C05384=1030.378,261.013,-119.631,170.542,45.453,158.713
C05385=1030.370,260.765,-119.601,170.539,45.453,158.712
C05386=1030.364,260.517,-119.572,170.535,45.454,158.712
C05387=1030.357,260.269,-119.542,170.532,45.455,158.712
C05388=1030.351,260.021,-119.513,170.528,45.456,158.712
C05389=1030.344,259.773,-119.483,170.525,45.457,158.712
C05390=1030.337,259.524,-119.453,170.521,45.457,158.711
C05391=1030.330,259.277,-119.424,170.518,45.458,158.711
C05392=1030.323,259.028,-119.395,170.513,45.459,158.711
C05393=1030.316,258.780,-119.366,170.510,45.460,158.711
C05394=1030.309,258.531,-119.336,170.506,45.461,158.711
C05395=1030.303,258.283,-119.307,170.503,45.461,158.710
C05396=1030.295,258.035,-119.277,170.499,45.462,158.710
C05397=1030.289,257.787,-119.248,170.496,45.463,158.710
C05398=1030.282,257.538,-119.219,170.492,45.464,158.710
C05399=1030.275,257.291,-119.189,170.489,45.465,158.710
C05400=1030.269,257.042,-119.159,170.485,45.466,158.709
C05401=1030.262,256.794,-119.130,170.482,45.466,158.709
C05402=1030.255,256.547,-119.101,170.478,45.467,158.709
C05403=1030.248,256.298,-119.072,170.475,45.468,158.709
C05404=1030.242,256.050,-119.043,170.471,45.469,158.709
C05405=1030.235,255.802,-119.013,170.468,45.470,158.709
C05406=1030.229,255.553,-118.984,170.465,45.470,158.708
C05407=1030.221,255.305,-118.955,170.461,45.471,158.708
C05408=1030.215,255.057,-118.926,170.458,45.472,158.708
C05409=1030.208,254.809,-118.896,170.454,45.473,158.708
C05410=1030.201,254.560,-118.867,170.451,45.474,158.708
C05411=1030.195,254.312,-118.838,170.447,45.475,158.708
C05412=1030.187,254.064,-118.809,170.444,45.476,158.707
C05413=1030.181,253.816,-118.780,170.440,45.477,158.707
C05414=1030.175,253.568,-118.750,170.437,45.478,158.707
C05415=1030.168,253.319,-118.721,170.434,45.478,158.707
C05416=1030.162,253.071,-118.691,170.430,45.479,158.707
C05417=1030.155,252.823,-118.663,170.427,45.480,158.706
C05418=1030.148,252.575,-118.634,170.423,45.481,158.706
C05419=1030.141,252.326,-118.605,170.420,45.482,158.706
C05420=1030.135,252.078,-118.576,170.417,45.483,158.706
C05421=1030.128,251.830,-118.545,170.413,45.484,158.706
C05422=1030.121,251.582,-118.517,170.410,45.484,158.706
C05423=1030.115,251.334,-118.488,170.406,45.485,158.705
C05424=1030.108,251.085,-118.459,170.403,45.486,158.705
C05425=1030.102,250.837,-118.429,170.400,45.487,158.705
C05426=1030.095,250.589,-118.400,170.396,45.488,158.705
C05427=1030.088,250.341,-118.372,170.393,45.489,158.705
C05428=1030.082,250.092,-118.343,170.389,45.490,158.705
C05429=1030.075,249.844,-118.314,170.386,45.491,158.704
C05430=1030.069,249.596,-118.284,170.383,45.491,158.704
C05431=1030.059,249.229,-118.242,170.378,45.493,158.704
C05432=1030.049,248.861,-118.199,170.373,45.494,158.704
C05433=1030.040,248.494,-118.155,170.368,45.496,158.704
C05434=1030.030,248.127,-118.113,170.363,45.497,158.703
C05435=1030.024,247.879,-118.084,170.360,45.497,158.703
C05436=1030.017,247.629,-118.055,170.356,45.499,158.703
C05437=1030.010,247.382,-118.027,170.353,45.500,158.703
C05438=1030.004,247.134,-117.998,170.350,45.500,158.703
C05439=1029.998,246.885,-117.969,170.346,45.501,158.702
C05440=1029.991,246.637,-117.940,170.343,45.503,158.702
C05441=1029.985,246.388,-117.910,170.340,45.503,158.702
C05442=1029.978,246.141,-117.882,170.336,45.504,158.702
C05443=1029.971,245.892,-117.853,170.333,45.505,158.702
C05444=1029.965,245.644,-117.824,170.330,45.506,158.702
C05445=1029.959,245.396,-117.795,170.326,45.507,158.702
C05446=1029.952,245.148,-117.767,170.323,45.508,158.702
C05447=1029.945,244.899,-117.737,170.320,45.509,158.701
C05448=1029.939,244.651,-117.708,170.316,45.510,158.701
C05449=1029.933,244.403,-117.679,170.313,45.511,158.701
C05450=1029.926,244.154,-117.652,170.310,45.512,158.701
C05451=1029.920,243.906,-117.623,170.306,45.513,158.701
C05452=1029.913,243.658,-117.594,170.303,45.514,158.701
C05453=1029.907,243.410,-117.566,170.300,45.515,158.701
C05454=1029.899,243.161,-117.537,170.297,45.516,158.700
C05455=1029.893,242.913,-117.508,170.294,45.517,158.700
C05456=1029.886,242.664,-117.480,170.291,45.518,158.700
C05457=1029.880,242.416,-117.451,170.287,45.519,158.700
C05458=1029.874,242.168,-117.423,170.284,45.520,158.700
C05459=1029.867,241.920,-117.394,170.281,45.521,158.700
C05460=1029.860,241.672,-117.366,170.277,45.522,158.700
C05461=1029.854,241.423,-117.338,170.274,45.524,158.700
C05462=1029.847,241.175,-117.309,170.271,45.524,158.699
C05463=1029.841,240.926,-117.281,170.267,45.525,158.699
C05464=1029.834,240.678,-117.252,170.264,45.527,158.699
C05465=1029.828,240.429,-117.224,170.261,45.527,158.699
C05466=1029.821,240.181,-117.195,170.259,45.529,158.699
C05467=1029.814,239.933,-117.168,170.254,45.530,158.699
C05468=1029.808,239.685,-117.139,170.252,45.531,158.699
C05469=1029.801,239.436,-117.111,170.249,45.532,158.699
C05470=1029.794,239.189,-117.082,170.245,45.533,158.699
C05471=1029.788,238.940,-117.055,170.242,45.535,158.699
C05472=1029.781,238.692,-117.026,170.239,45.535,158.698
C05473=1029.775,238.444,-116.998,170.235,45.537,158.698
C05474=1029.768,238.195,-116.970,170.232,45.538,158.698
C05475=1029.761,237.947,-116.942,170.229,45.539,158.698
C05476=1029.754,237.698,-116.913,170.225,45.540,158.698
C05477=1029.748,237.449,-116.885,170.223,45.541,158.698
C05478=1029.741,237.202,-116.857,170.220,45.543,158.698
C05479=1029.734,236.953,-116.829,170.216,45.543,158.698
C05480=1029.727,236.705,-116.801,170.213,45.545,158.698
C05481=1029.722,236.456,-116.773,170.210,45.546,158.698
C05482=1029.715,236.208,-116.745,170.207,45.547,158.698
C05483=1029.708,235.960,-116.717,170.203,45.548,158.697
C05484=1029.701,235.711,-116.689,170.200,45.549,158.697
C05485=1029.694,235.463,-116.661,170.198,45.550,158.697
C05486=1029.687,235.215,-116.633,170.194,45.552,158.697
C05487=1029.678,234.842,-116.591,170.189,45.554,158.697
C05488=1029.668,234.468,-116.550,170.184,45.556,158.697
C05489=1029.658,234.095,-116.507,170.181,45.557,158.697
C05490=1029.649,233.721,-116.465,170.176,45.559,158.697
C05491=1029.642,233.473,-116.437,170.172,45.560,158.697
C05492=1029.635,233.225,-116.409,170.169,45.561,158.697
C05493=1029.629,232.976,-116.382,170.166,45.563,158.697
C05494=1029.622,232.728,-116.354,170.163,45.563,158.696
C05495=1029.615,232.480,-116.325,170.159,45.565,158.696
C05496=1029.608,232.231,-116.298,170.157,45.566,158.696
C05497=1029.602,231.983,-116.269,170.154,45.567,158.696
C05498=1029.596,231.734,-116.242,170.151,45.568,158.696
C05499=1029.589,231.486,-116.214,170.147,45.570,158.696
C05500=1029.582,231.237,-116.186,170.144,45.571,158.696
C05501=1029.576,230.989,-116.158,170.141,45.572,158.696
C05502=1029.570,230.741,-116.131,170.138,45.573,158.696
C05503=1029.563,230.493,-116.103,170.135,45.575,158.696
C05504=1029.556,230.244,-116.076,170.132,45.576,158.696
C05505=1029.550,229.996,-116.048,170.129,45.577,158.696
C05506=1029.543,229.747,-116.020,170.126,45.578,158.696
C05507=1029.536,229.499,-115.992,170.122,45.580,158.696
C05508=1029.530,229.250,-115.965,170.120,45.581,158.696
C05509=1029.523,229.002,-115.937,170.117,45.583,158.696
C05510=1029.516,228.754,-115.909,170.114,45.583,158.695
C05511=1029.509,228.505,-115.882,170.110,45.585,158.695
C05512=1029.503,228.257,-115.854,170.107,45.586,158.695
C05513=1029.497,228.008,-115.827,170.104,45.588,158.695
C05514=1029.490,227.760,-115.799,170.102,45.589,158.695
C05515=1029.484,227.511,-115.772,170.098,45.590,158.695
C05516=1029.477,227.263,-115.744,170.095,45.591,158.695
C05517=1029.470,227.015,-115.716,170.092,45.593,158.695
C05518=1029.463,226.766,-115.689,170.089,45.594,158.695
C05519=1029.457,226.518,-115.662,170.085,45.596,158.695
C05520=1029.450,226.270,-115.635,170.083,45.597,158.695
C05521=1029.444,226.021,-115.607,170.080,45.598,158.695
C05522=1029.436,225.773,-115.580,170.077,45.600,158.695
C05523=1029.430,225.524,-115.553,170.073,45.601,158.695
C05524=1029.423,225.276,-115.525,170.071,45.603,158.695
C05525=1029.417,225.028,-115.498,170.068,45.604,158.695
C05526=1029.410,224.779,-115.471,170.065,45.605,158.695
C05527=1029.403,224.531,-115.444,170.061,45.607,158.695
C05528=1029.397,224.282,-115.416,170.059,45.608,158.695
C05529=1029.390,224.033,-115.389,170.056,45.610,158.695
C05530=1029.383,223.785,-115.362,170.053,45.611,158.695
C05531=1029.377,223.537,-115.334,170.049,45.612,158.695
C05532=1029.370,223.288,-115.307,170.046,45.614,158.695
C05533=1029.364,223.040,-115.280,170.043,45.615,158.694
C05534=1029.356,222.792,-115.252,170.041,45.616,158.694
C05535=1029.351,222.543,-115.226,170.038,45.617,158.694
C05536=1029.344,222.295,-115.198,170.034,45.619,158.694
C05537=1029.338,222.046,-115.171,170.031,45.620,158.694
C05538=1029.330,221.798,-115.144,170.029,45.621,158.694
C05539=1029.323,221.549,-115.116,170.026,45.623,158.694
C05540=1029.318,221.301,-115.090,170.023,45.624,158.694
C05541=1029.311,221.052,-115.062,170.019,45.626,158.694
C05542=1029.304,220.804,-115.035,170.016,45.627,158.694
C05543=1029.294,220.423,-114.994,170.012,45.630,158.694
C05544=1029.284,220.042,-114.951,170.007,45.631,158.694
C05545=1029.274,219.661,-114.910,170.004,45.634,158.694
C05546=1029.264,219.279,-114.869,169.999,45.636,158.694
C05547=1029.257,219.032,-114.842,169.995,45.638,158.694
C05548=1029.251,218.783,-114.815,169.993,45.639,158.694
C05549=1029.244,218.534,-114.788,169.990,45.640,158.694
C05550=1029.237,218.286,-114.761,169.987,45.642,158.694
C05551=1029.230,218.038,-114.735,169.984,45.643,158.694
C05552=1029.224,217.789,-114.707,169.980,45.645,158.694
C05553=1029.217,217.540,-114.681,169.978,45.647,158.694
C05554=1029.211,217.292,-114.654,169.975,45.648,158.694
C05555=1029.203,217.044,-114.627,169.972,45.649,158.694
C05556=1029.197,216.795,-114.600,169.970,45.651,158.694
C05557=1029.191,216.547,-114.574,169.966,45.652,158.694
C05558=1029.183,216.298,-114.547,169.963,45.654,158.694
C05559=1029.177,216.050,-114.520,169.961,45.656,158.694
C05560=1029.170,215.802,-114.493,169.958,45.657,158.694
C05561=1029.164,215.552,-114.466,169.955,45.658,158.694
C05562=1029.156,215.304,-114.439,169.951,45.660,158.694
C05563=1029.151,215.056,-114.413,169.948,45.661,158.694
C05564=1029.144,214.807,-114.386,169.946,45.663,158.694
C05565=1029.137,214.558,-114.359,169.943,45.665,158.694
C05566=1029.131,214.310,-114.333,169.940,45.666,158.694
C05567=1029.124,214.062,-114.305,169.938,45.667,158.694
C05568=1029.117,213.813,-114.279,169.934,45.669,158.694
C05569=1029.110,213.565,-114.253,169.931,45.671,158.694
C05570=1029.104,213.316,-114.226,169.929,45.672,158.694
C05571=1029.098,213.068,-114.200,169.926,45.674,158.694
C05572=1029.091,212.819,-114.172,169.923,45.675,158.694
C05573=1029.084,212.571,-114.146,169.920,45.676,158.694
C05574=1029.078,212.322,-114.119,169.917,45.679,158.694
C05575=1029.071,212.073,-114.093,169.914,45.680,158.694
C05576=1029.065,211.825,-114.066,169.911,45.681,158.694
C05577=1029.058,211.576,-114.040,169.908,45.683,158.694
C05578=1029.051,211.328,-114.013,169.906,45.685,158.695
C05579=1029.045,211.080,-113.986,169.903,45.686,158.695
C05580=1029.038,210.831,-113.959,169.900,45.687,158.695
C05581=1029.032,210.583,-113.933,169.897,45.689,158.694
C05582=1029.025,210.334,-113.906,169.894,45.691,158.695
C05583=1029.018,210.086,-113.880,169.891,45.692,158.695
C05584=1029.011,209.837,-113.854,169.889,45.694,158.695
C05585=1029.005,209.589,-113.827,169.886,45.696,158.695
C05586=1028.998,209.340,-113.801,169.883,45.697,158.695
C05587=1028.991,209.091,-113.774,169.881,45.698,158.695
C05588=1028.985,208.843,-113.748,169.877,45.701,158.695
C05589=1028.978,208.594,-113.721,169.874,45.702,158.695
C05590=1028.972,208.346,-113.695,169.872,45.703,158.695
C05591=1028.965,208.097,-113.669,169.869,45.705,158.695
C05592=1028.958,207.849,-113.643,169.866,45.707,158.695
C05593=1028.951,207.601,-113.616,169.864,45.708,158.695
C05594=1028.946,207.352,-113.590,169.861,45.710,158.695
C05595=1028.938,207.103,-113.564,169.857,45.712,158.695
C05596=1028.932,206.855,-113.538,169.855,45.714,158.695
C05597=1028.925,206.606,-113.512,169.852,45.715,158.695
C05598=1028.918,206.358,-113.486,169.849,45.716,158.695
C05599=1028.908,205.982,-113.446,169.845,45.720,158.695
C05600=1028.899,205.606,-113.406,169.840,45.722,158.695
C05601=1028.888,205.231,-113.367,169.837,45.724,158.695
C05602=1028.878,204.855,-113.327,169.832,45.727,158.695
C05603=1028.852,203.809,-113.223,169.464,45.624,158.634
C05604=1028.846,203.560,-113.198,169.460,45.626,158.634
C05605=1028.841,203.311,-113.174,169.456,45.628,158.634
C05606=1028.835,203.063,-113.149,169.452,45.631,158.634
C05607=1028.829,202.814,-113.124,169.449,45.633,158.634
C05608=1028.822,202.566,-113.100,169.444,45.636,158.634
C05609=1028.817,202.317,-113.075,169.441,45.638,158.635
C05610=1028.811,202.069,-113.050,169.437,45.641,158.635
C05611=1028.805,201.819,-113.025,169.433,45.643,158.635
C05612=1028.799,201.570,-113.001,169.430,45.646,158.635
C05613=1028.793,201.322,-112.976,169.426,45.648,158.635
C05614=1028.787,201.073,-112.952,169.423,45.650,158.635
C05615=1028.781,200.825,-112.927,169.418,45.653,158.635
C05616=1028.775,200.576,-112.902,169.415,45.656,158.635
C05617=1028.769,200.327,-112.878,169.411,45.658,158.635
C05618=1028.763,200.078,-112.854,169.407,45.660,158.635
C05619=1028.757,199.830,-112.829,169.403,45.663,158.636
C05620=1028.751,199.581,-112.805,169.400,45.666,158.636
C05621=1028.745,199.332,-112.780,169.395,45.668,158.636
C05622=1028.739,199.083,-112.756,169.392,45.671,158.636
C05623=1028.733,198.834,-112.732,169.389,45.673,158.636
C05624=1028.727,198.585,-112.708,169.384,45.676,158.636
C05625=1028.721,198.338,-112.683,169.381,45.679,158.636
C05626=1028.714,198.089,-112.659,169.377,45.682,158.637
C05627=1028.709,197.839,-112.634,169.374,45.684,158.637
C05628=1028.703,197.591,-112.611,169.370,45.687,158.637
C05629=1028.697,197.342,-112.586,169.366,45.689,158.637
C05630=1028.691,197.093,-112.562,169.363,45.692,158.637
C05631=1028.685,196.844,-112.538,169.358,45.695,158.637
C05632=1028.679,196.596,-112.514,169.355,45.697,158.637
C05633=1028.672,196.347,-112.490,169.352,45.700,158.637
C05634=1028.667,196.098,-112.466,169.348,45.703,158.638
C05635=1028.660,195.849,-112.442,169.344,45.705,158.638
C05636=1028.655,195.601,-112.418,169.340,45.707,158.638
C05637=1028.648,195.352,-112.394,169.337,45.710,158.638
C05638=1028.643,195.103,-112.369,169.333,45.712,158.638
C05639=1028.636,194.854,-112.345,169.329,45.716,158.638
C05640=1028.631,194.606,-112.321,169.326,45.718,158.638
C05641=1028.624,194.357,-112.297,169.322,45.721,158.639
C05642=1028.619,194.108,-112.273,169.319,45.723,158.639
C05643=1028.612,193.859,-112.249,169.315,45.726,158.639
C05644=1028.606,193.611,-112.225,169.311,45.729,158.639
C05645=1028.601,193.362,-112.201,169.308,45.731,158.639
C05646=1028.594,193.113,-112.177,169.305,45.734,158.639
C05647=1028.589,192.865,-112.153,169.301,45.736,158.640
C05648=1028.582,192.616,-112.129,169.297,45.740,158.640
C05649=1028.577,192.366,-112.105,169.293,45.742,158.640
C05650=1028.571,192.117,-112.081,169.290,45.745,158.640
C05651=1028.565,191.869,-112.057,169.286,45.747,158.640
C05652=1028.559,191.621,-112.033,169.283,45.750,158.640
C05653=1028.553,191.372,-112.009,169.279,45.752,158.640
C05654=1028.548,191.123,-111.985,169.275,45.755,158.641
C05655=1028.542,190.874,-111.962,169.272,45.758,158.641
C05656=1028.536,190.625,-111.937,169.269,45.760,158.641
C05657=1028.530,190.377,-111.914,169.265,45.763,158.641
C05658=1028.523,190.128,-111.889,169.261,45.766,158.641
C05659=1028.518,189.879,-111.865,169.258,45.769,158.641
C05660=1028.512,189.630,-111.842,169.254,45.771,158.641
C05661=1028.506,189.381,-111.818,169.251,45.774,158.642
C05662=1028.500,189.133,-111.794,169.247,45.776,158.642
C05663=1028.495,188.884,-111.770,169.244,45.779,158.642
C05664=1028.488,188.600,-111.743,169.240,45.782,158.642
C05665=1028.482,188.317,-111.716,169.235,45.785,158.642
C05666=1028.474,188.034,-111.689,169.232,45.788,158.643
C05667=1028.468,187.751,-111.662,169.228,45.791,158.643
C05668=1028.463,187.502,-111.638,169.224,45.794,158.643
C05669=1028.456,187.253,-111.614,169.221,45.797,158.643
C05670=1028.450,187.005,-111.590,169.218,45.799,158.643
C05671=1028.445,186.756,-111.567,169.213,45.802,158.643
C05672=1028.439,186.507,-111.543,169.210,45.804,158.643
C05673=1028.434,186.257,-111.519,169.207,45.807,158.644
C05674=1028.428,186.009,-111.496,169.203,45.810,158.644
C05675=1028.422,185.761,-111.472,169.200,45.812,158.644
C05676=1028.417,185.512,-111.448,169.197,45.815,158.644
C05677=1028.410,185.263,-111.424,169.193,45.817,158.644
C05678=1028.405,185.014,-111.401,169.190,45.820,158.644
C05679=1028.399,184.765,-111.377,169.186,45.823,158.645
C05680=1028.393,184.517,-111.353,169.183,45.826,158.645
C05681=1028.388,184.268,-111.330,169.180,45.829,158.645
C05682=1028.381,184.019,-111.306,169.176,45.831,158.645
C05683=1028.376,183.770,-111.282,169.172,45.834,158.645
C05684=1028.370,183.521,-111.259,169.168,45.836,158.645
C05685=1028.364,183.272,-111.236,169.165,45.839,158.646
C05686=1028.359,183.024,-111.211,169.162,45.842,158.646
C05687=1028.353,182.775,-111.189,169.158,45.844,158.646
C05688=1028.347,182.526,-111.165,169.155,45.847,158.646
C05689=1028.341,182.277,-111.142,169.152,45.850,158.646
C05690=1028.335,182.028,-111.119,169.149,45.853,158.647
C05691=1028.329,181.780,-111.096,169.145,45.856,158.647
C05692=1028.323,181.530,-111.073,169.141,45.859,158.647
C05693=1028.317,181.282,-111.049,169.138,45.862,158.647
C05694=1028.311,181.033,-111.026,169.135,45.865,158.647
C05695=1028.304,180.784,-111.004,169.131,45.868,158.648
C05696=1028.298,180.535,-110.981,169.128,45.871,158.648
C05697=1028.292,180.286,-110.957,169.125,45.874,158.648
C05698=1028.286,180.037,-110.934,169.121,45.876,158.648
C05699=1028.280,179.789,-110.911,169.118,45.879,158.648
C05700=1028.274,179.540,-110.889,169.114,45.882,158.649
C05701=1028.268,179.290,-110.865,169.111,45.885,158.649
C05702=1028.262,179.041,-110.843,169.107,45.888,158.649
C05703=1028.256,178.793,-110.820,169.104,45.891,158.649
C05704=1028.250,178.544,-110.796,169.101,45.894,158.650
C05705=1028.244,178.296,-110.774,169.098,45.897,158.650
C05706=1028.238,178.047,-110.751,169.094,45.900,158.650
C05707=1028.232,177.797,-110.727,169.091,45.903,158.650
C05708=1028.226,177.548,-110.704,169.088,45.906,158.650
C05709=1028.219,177.300,-110.682,169.085,45.908,158.651
C05710=1028.214,177.051,-110.659,169.080,45.912,158.651
C05711=1028.208,176.802,-110.636,169.077,45.915,158.651
C05712=1028.202,176.553,-110.613,169.074,45.917,158.651
C05713=1028.197,176.304,-110.590,169.071,45.920,158.652
C05714=1028.190,176.056,-110.568,169.067,45.923,158.652
C05715=1028.184,175.807,-110.545,169.064,45.926,158.652
C05716=1028.178,175.557,-110.522,169.061,45.929,158.652
C05717=1028.172,175.308,-110.499,169.058,45.932,158.652
C05718=1028.166,175.060,-110.476,169.054,45.934,158.653
C05719=1028.160,174.811,-110.453,169.051,45.937,158.653
C05720=1028.154,174.562,-110.430,169.048,45.940,158.653
C05721=1028.149,174.313,-110.407,169.044,45.943,158.653
C05722=1028.142,174.064,-110.385,169.041,45.946,158.653
C05723=1028.136,173.815,-110.362,169.038,45.949,158.654
C05724=1028.131,173.566,-110.339,169.035,45.952,158.654
C05725=1028.125,173.318,-110.316,169.031,45.955,158.654
C05726=1028.118,173.069,-110.294,169.028,45.958,158.654
C05727=1028.113,172.820,-110.271,169.025,45.961,158.655
C05728=1028.106,172.536,-110.245,169.021,45.965,158.655
C05729=1028.099,172.253,-110.219,169.018,45.968,158.655
C05730=1028.093,171.969,-110.193,169.013,45.971,158.655
C05731=1028.086,171.685,-110.168,169.009,45.975,158.656
C05732=1028.080,171.436,-110.145,169.006,45.978,158.656
C05733=1028.074,171.187,-110.122,169.003,45.980,158.656
C05734=1028.068,170.939,-110.099,169.001,45.983,158.656
C05735=1028.063,170.690,-110.077,168.997,45.986,158.657
C05736=1028.057,170.441,-110.055,168.994,45.989,158.657
C05737=1028.052,170.192,-110.032,168.991,45.992,158.657
C05738=1028.045,169.943,-110.009,168.988,45.995,158.657
C05739=1028.039,169.695,-109.986,168.984,45.998,158.658
C05740=1028.034,169.446,-109.963,168.981,46.001,158.658
C05741=1028.028,169.196,-109.941,168.978,46.004,158.658
C05742=1028.022,168.948,-109.919,168.975,46.007,158.658
C05743=1028.016,168.699,-109.896,168.971,46.010,158.658
C05744=1028.010,168.450,-109.873,168.968,46.013,158.659
C05745=1028.004,168.201,-109.851,168.965,46.015,158.659
C05746=1027.998,167.952,-109.828,168.961,46.018,158.659
C05747=1027.993,167.703,-109.805,168.958,46.021,158.659
C05748=1027.987,167.454,-109.782,168.955,46.024,158.659
C05749=1027.981,167.205,-109.761,168.952,46.027,158.660
C05750=1027.976,166.956,-109.738,168.948,46.030,158.660
C05751=1027.970,166.708,-109.715,168.945,46.032,158.660
C05752=1027.964,166.458,-109.693,168.942,46.035,158.660
C05753=1027.958,166.209,-109.671,168.940,46.038,158.661
C05754=1027.952,165.961,-109.648,168.936,46.041,158.661
C05755=1027.947,165.711,-109.625,168.933,46.044,158.661
C05756=1027.941,165.463,-109.604,168.930,46.047,158.661
C05757=1027.935,165.214,-109.581,168.927,46.050,158.662
C05758=1027.930,164.965,-109.558,168.923,46.053,158.662
C05759=1027.924,164.716,-109.535,168.920,46.056,158.662
C05760=1027.918,164.467,-109.514,168.917,46.059,158.662
C05761=1027.912,164.218,-109.491,168.914,46.062,158.662
C05762=1027.907,163.970,-109.468,168.911,46.064,158.663
C05763=1027.901,163.720,-109.447,168.908,46.067,158.663
C05764=1027.895,163.471,-109.424,168.905,46.070,158.663
C05765=1027.890,163.222,-109.401,168.902,46.073,158.663
C05766=1027.884,162.973,-109.378,168.898,46.076,158.664
C05767=1027.878,162.725,-109.356,168.895,46.079,158.664
C05768=1027.873,162.476,-109.334,168.892,46.082,158.664
C05769=1027.867,162.227,-109.311,168.890,46.085,158.664
C05770=1027.861,161.978,-109.290,168.887,46.088,158.665
C05771=1027.856,161.729,-109.267,168.883,46.091,158.665
C05772=1027.850,161.480,-109.245,168.880,46.094,158.665
C05773=1027.844,161.231,-109.223,168.877,46.097,158.665
C05774=1027.838,160.982,-109.200,168.874,46.100,158.665
C05775=1027.833,160.734,-109.178,168.870,46.103,158.666
C05776=1027.828,160.484,-109.155,168.868,46.105,158.666
C05777=1027.821,160.235,-109.133,168.865,46.108,158.666
C05778=1027.816,159.986,-109.111,168.862,46.111,158.666
C05779=1027.811,159.737,-109.089,168.858,46.114,158.667
C05780=1027.805,159.488,-109.067,168.855,46.117,158.667
C05781=1027.799,159.239,-109.044,168.853,46.120,158.667
C05782=1027.793,158.990,-109.023,168.850,46.123,158.668
C05783=1027.787,158.742,-109.001,168.847,46.126,158.668
C05784=1027.782,158.492,-108.979,168.843,46.129,158.668
C05785=1027.776,158.243,-108.957,168.840,46.132,158.668
C05786=1027.769,157.994,-108.935,168.837,46.135,158.668
C05787=1027.764,157.746,-108.913,168.834,46.139,158.669
C05788=1027.758,157.497,-108.891,168.831,46.142,158.669
C05789=1027.752,157.247,-108.869,168.827,46.145,158.669
C05790=1027.746,156.998,-108.848,168.825,46.147,158.670
C05791=1027.740,156.750,-108.827,168.822,46.151,158.670
C05792=1027.733,156.465,-108.801,168.818,46.154,158.670
C05793=1027.726,156.182,-108.776,168.815,46.158,158.670
C05794=1027.720,155.897,-108.752,168.811,46.162,158.671
C05795=1027.713,155.614,-108.727,168.808,46.165,158.671
C05796=1027.708,155.364,-108.705,168.805,46.168,158.671
C05797=1027.702,155.115,-108.683,168.802,46.171,158.672
C05798=1027.696,154.866,-108.661,168.799,46.174,158.672
C05799=1027.690,154.618,-108.639,168.796,46.177,158.672
C05800=1027.684,154.369,-108.617,168.793,46.180,158.672
C05801=1027.678,154.119,-108.595,168.790,46.184,158.673
C05802=1027.673,153.871,-108.574,168.787,46.187,158.673
C05803=1027.666,153.622,-108.553,168.784,46.190,158.673
C05804=1027.661,153.372,-108.530,168.780,46.192,158.673
C05805=1027.655,153.124,-108.509,168.778,46.196,158.674
C05806=1027.649,152.874,-108.487,168.775,46.199,158.674
C05807=1027.643,152.625,-108.466,168.772,46.202,158.674
C05808=1027.638,152.377,-108.445,168.769,46.205,158.675
C05809=1027.631,152.128,-108.423,168.766,46.208,158.675
C05810=1027.625,151.878,-108.401,168.762,46.211,158.675
C05811=1027.620,151.630,-108.380,168.760,46.214,158.675
C05812=1027.613,151.381,-108.358,168.757,46.218,158.676
C05813=1027.607,151.131,-108.337,168.754,46.221,158.676
C05814=1027.603,150.883,-108.315,168.751,46.224,158.676
C05815=1027.596,150.633,-108.293,168.748,46.227,158.677
C05816=1027.591,150.385,-108.272,168.745,46.230,158.677
C05817=1027.585,150.136,-108.250,168.742,46.233,158.677
C05818=1027.578,149.887,-108.229,168.739,46.236,158.677
C05819=1027.573,149.637,-108.208,168.736,46.240,158.678
C05820=1027.567,149.388,-108.187,168.733,46.243,158.678
C05821=1027.561,149.140,-108.165,168.730,46.246,158.678
C05822=1027.555,148.890,-108.144,168.728,46.249,158.679
C05823=1027.549,148.641,-108.122,168.724,46.252,158.679
C05824=1027.544,148.393,-108.101,168.721,46.255,158.679
C05825=1027.537,148.144,-108.079,168.718,46.258,158.679
C05826=1027.532,147.895,-108.058,168.715,46.261,158.680
C05827=1027.526,147.645,-108.037,168.713,46.264,158.680
C05828=1027.520,147.397,-108.016,168.710,46.267,158.680
C05829=1027.514,147.148,-107.994,168.707,46.271,158.681
C05830=1027.508,146.898,-107.972,168.703,46.274,158.681
C05831=1027.503,146.650,-107.951,168.700,46.277,158.681
C05832=1027.497,146.400,-107.930,168.698,46.280,158.681
C05833=1027.491,146.151,-107.909,168.695,46.283,158.682
C05834=1027.485,145.902,-107.887,168.692,46.286,158.682
C05835=1027.480,145.653,-107.867,168.689,46.290,158.682
C05836=1027.474,145.404,-107.845,168.686,46.293,158.682
C05837=1027.468,145.155,-107.824,168.684,46.296,158.683
C05838=1027.461,144.906,-107.803,168.680,46.299,158.683
C05839=1027.455,144.657,-107.782,168.677,46.303,158.683
C05840=1027.450,144.408,-107.761,168.674,46.306,158.684
C05841=1027.444,144.158,-107.740,168.671,46.309,158.684
C05842=1027.438,143.910,-107.718,168.669,46.312,158.684
C05843=1027.432,143.661,-107.697,168.666,46.315,158.685
C05844=1027.426,143.412,-107.677,168.663,46.319,158.685
C05845=1027.420,143.163,-107.655,168.660,46.322,158.685
C05846=1027.414,142.914,-107.634,168.657,46.324,158.685
C05847=1027.409,142.664,-107.613,168.654,46.328,158.686
C05848=1027.403,142.416,-107.592,168.651,46.331,158.686
C05849=1027.396,142.166,-107.571,168.648,46.335,158.686
C05850=1027.391,141.918,-107.550,168.646,46.337,158.687
C05851=1027.385,141.668,-107.529,168.643,46.340,158.687
C05852=1027.379,141.419,-107.508,168.640,46.344,158.687
C05853=1027.373,141.170,-107.486,168.637,46.347,158.688
C05854=1027.368,140.921,-107.466,168.633,46.350,158.688
C05855=1027.362,140.673,-107.445,168.631,46.353,158.688
C05856=1027.355,140.388,-107.421,168.627,46.357,158.688
C05857=1027.349,140.103,-107.397,168.625,46.361,158.689
C05858=1027.342,139.819,-107.373,168.621,46.364,158.689
C05859=1027.335,139.535,-107.349,168.618,46.368,158.689
C05860=1027.330,139.286,-107.328,168.615,46.371,158.690
C05861=1027.323,139.037,-107.307,168.612,46.374,158.690
C05862=1027.318,138.788,-107.287,168.609,46.377,158.690
C05863=1027.312,138.539,-107.265,168.607,46.381,158.691
C05864=1027.306,138.290,-107.245,168.604,46.384,158.691
C05865=1027.300,138.040,-107.224,168.601,46.387,158.691
C05866=1027.294,137.792,-107.203,168.598,46.390,158.692
C05867=1027.288,137.543,-107.183,168.596,46.394,158.692
C05868=1027.282,137.294,-107.161,168.592,46.397,158.692
C05869=1027.277,137.044,-107.141,168.589,46.400,158.693
C05870=1027.270,136.795,-107.120,168.587,46.403,158.693
C05871=1027.265,136.546,-107.099,168.584,46.407,158.693
C05872=1027.259,136.297,-107.079,168.581,46.410,158.693
C05873=1027.253,136.048,-107.058,168.578,46.413,158.694
C05874=1027.247,135.799,-107.037,168.576,46.416,158.694
C05875=1027.241,135.550,-107.017,168.573,46.420,158.694
C05876=1027.235,135.301,-106.996,168.570,46.423,158.695
C05877=1027.229,135.052,-106.975,168.567,46.426,158.695
C05878=1027.223,134.803,-106.954,168.565,46.429,158.695
C05879=1027.217,134.554,-106.935,168.561,46.432,158.696
C05880=1027.211,134.304,-106.914,168.558,46.436,158.696
C05881=1027.206,134.056,-106.892,168.555,46.439,158.696
C05882=1027.200,133.807,-106.872,168.553,46.442,158.697
C05883=1027.194,133.557,-106.851,168.550,46.445,158.697
C05884=1027.188,133.308,-106.831,168.547,46.449,158.697
C05885=1027.182,133.060,-106.810,168.545,46.452,158.697
C05886=1027.176,132.810,-106.790,168.542,46.455,158.698
C05887=1027.171,132.561,-106.769,168.539,46.458,158.698
C05888=1027.165,132.312,-106.749,168.536,46.462,158.698
C05889=1027.159,132.062,-106.728,168.534,46.465,158.699
C05890=1027.152,131.814,-106.708,168.531,46.468,158.699
C05891=1027.147,131.565,-106.687,168.527,46.471,158.699
C05892=1027.141,131.315,-106.666,168.525,46.475,158.700
C05893=1027.135,131.066,-106.646,168.522,46.478,158.700
C05894=1027.130,130.817,-106.626,168.519,46.482,158.700
C05895=1027.124,130.568,-106.606,168.517,46.484,158.701
C05896=1027.118,130.319,-106.585,168.514,46.488,158.701
C05897=1027.112,130.070,-106.564,168.511,46.491,158.701
C05898=1027.106,129.822,-106.544,168.508,46.495,158.702
C05899=1027.099,129.572,-106.524,168.506,46.497,158.702
C05900=1027.093,129.323,-106.504,168.503,46.501,158.702
C05901=1027.088,129.074,-106.483,168.500,46.505,158.703
C05902=1027.082,128.825,-106.463,168.497,46.508,158.703
C05903=1027.076,128.575,-106.444,168.495,46.511,158.703
C05904=1027.070,128.326,-106.424,168.492,46.515,158.704
C05905=1027.063,128.077,-106.404,168.489,46.518,158.704
C05906=1027.058,127.828,-106.383,168.486,46.521,158.704
C05907=1027.052,127.579,-106.363,168.484,46.525,158.705
C05908=1027.045,127.329,-106.343,168.480,46.528,158.705
C05909=1027.039,127.081,-106.323,168.478,46.532,158.705
C05910=1027.034,126.831,-106.302,168.475,46.534,158.705
C05911=1027.028,126.583,-106.282,168.472,46.538,158.706
C05912=1027.022,126.333,-106.262,168.469,46.542,158.706
C05913=1027.016,126.084,-106.242,168.466,46.545,158.706
C05914=1027.010,125.835,-106.222,168.464,46.548,158.707
C05915=1027.004,125.587,-106.202,168.461,46.552,158.707
C05916=1026.998,125.336,-106.182,168.458,46.555,158.707
C05917=1026.992,125.087,-106.162,168.456,46.558,158.708
C05918=1026.986,124.839,-106.142,168.453,46.561,158.708
C05919=1026.980,124.590,-106.122,168.450,46.565,158.708
C05920=1026.974,124.305,-106.099,168.447,46.569,158.709
C05921=1026.966,124.021,-106.076,168.444,46.572,158.709
C05922=1026.959,123.736,-106.053,168.441,46.576,158.710
C05923=1026.953,123.452,-106.030,168.437,46.580,158.710
C05924=1026.947,123.203,-106.010,168.435,46.583,158.710
C05925=1026.941,122.954,-105.990,168.432,46.587,158.711
C05926=1026.935,122.704,-105.971,168.429,46.590,158.711
C05927=1026.929,122.455,-105.950,168.427,46.593,158.711
C05928=1026.923,122.206,-105.930,168.424,46.596,158.712
C05929=1026.917,121.957,-105.910,168.421,46.600,158.712
C05930=1026.911,121.708,-105.890,168.419,46.603,158.712
C05931=1026.906,121.459,-105.871,168.416,46.607,158.713
C05932=1026.900,121.209,-105.850,168.413,46.610,158.713
C05933=1026.894,120.960,-105.830,168.411,46.613,158.713
C05934=1026.888,120.711,-105.810,168.408,46.617,158.714
C05935=1026.882,120.462,-105.791,168.405,46.620,158.714
C05936=1026.876,120.213,-105.771,168.403,46.623,158.714
C05937=1026.870,119.964,-105.751,168.400,46.626,158.714
C05938=1026.864,119.715,-105.730,168.398,46.630,158.715
C05939=1026.859,119.465,-105.711,168.395,46.633,158.715
C05940=1026.853,119.216,-105.691,168.391,46.636,158.715
C05941=1026.847,118.968,-105.671,168.390,46.640,158.716
C05942=1026.841,118.718,-105.652,168.386,46.643,158.716
C05943=1026.835,118.469,-105.632,168.383,46.647,158.716
C05944=1026.830,118.220,-105.611,168.381,46.649,158.717
C05945=1026.824,117.971,-105.592,168.378,46.653,158.717
C05946=1026.818,117.722,-105.572,168.375,46.656,158.717
C05947=1026.811,117.472,-105.551,168.373,46.659,158.718
C05948=1026.806,117.223,-105.532,168.370,46.663,158.718
C05949=1026.800,116.974,-105.512,168.368,46.666,158.718
C05950=1026.795,116.725,-105.492,168.365,46.670,158.719
C05951=1026.789,116.476,-105.472,168.362,46.673,158.719
C05952=1026.783,116.227,-105.453,168.360,46.676,158.719
C05953=1026.777,115.978,-105.433,168.357,46.679,158.720
C05954=1026.771,115.729,-105.413,168.355,46.683,158.720
C05955=1026.765,115.480,-105.393,168.352,46.686,158.720
C05956=1026.759,115.230,-105.374,168.349,46.689,158.721
C05957=1026.754,114.981,-105.354,168.346,46.692,158.721
C05958=1026.749,114.732,-105.334,168.344,46.696,158.721
C05959=1026.743,114.483,-105.314,168.341,46.698,158.722
C05960=1026.737,114.234,-105.294,168.338,46.702,158.722
C05961=1026.731,113.985,-105.275,168.336,46.705,158.722
C05962=1026.725,113.736,-105.255,168.333,46.709,158.723
C05963=1026.720,113.486,-105.235,168.330,46.712,158.723
C05964=1026.713,113.237,-105.215,168.328,46.715,158.723
C05965=1026.708,112.987,-105.196,168.325,46.718,158.723
C05966=1026.702,112.738,-105.176,168.323,46.722,158.724
C05967=1026.696,112.489,-105.157,168.320,46.725,158.724
C05968=1026.690,112.240,-105.137,168.317,46.728,158.724
C05969=1026.684,111.991,-105.117,168.315,46.732,158.725
C05970=1026.678,111.742,-105.099,168.312,46.735,158.725
C05971=1026.672,111.493,-105.079,168.309,46.738,158.725
C05972=1026.666,111.243,-105.060,168.307,46.742,158.726
C05973=1026.660,110.995,-105.040,168.304,46.745,158.726
C05974=1026.654,110.745,-105.020,168.302,46.748,158.727
C05975=1026.649,110.496,-105.001,168.299,46.752,158.727
C05976=1026.643,110.247,-104.981,168.296,46.755,158.727
C05977=1026.637,109.997,-104.962,168.294,46.759,158.728
C05978=1026.631,109.748,-104.943,168.291,46.762,158.728
C05979=1026.625,109.499,-104.923,168.288,46.765,158.728
C05980=1026.619,109.250,-104.904,168.286,46.769,158.729
C05981=1026.613,109.001,-104.885,168.283,46.772,158.729
C05982=1026.607,108.751,-104.866,168.281,46.775,158.729
C05983=1026.601,108.503,-104.846,168.278,46.779,158.730
C05984=1026.594,108.218,-104.824,168.275,46.783,158.730
C05985=1026.588,107.933,-104.803,168.272,46.787,158.730
C05986=1026.580,107.649,-104.781,168.268,46.791,158.731
C05987=1026.573,107.364,-104.759,168.265,46.795,158.731
C05988=1026.567,107.115,-104.739,168.263,46.798,158.732
C05989=1026.562,106.865,-104.720,168.260,46.801,158.732
C05990=1026.555,106.616,-104.701,168.257,46.805,158.732
C05991=1026.550,106.367,-104.682,168.255,46.808,158.733
C05992=1026.544,106.118,-104.662,168.252,46.811,158.733
C05993=1026.537,105.869,-104.644,168.250,46.815,158.733
C05994=1026.532,105.620,-104.625,168.247,46.819,158.734
C05995=1026.526,105.371,-104.605,168.244,46.822,158.734
C05996=1026.520,105.122,-104.587,168.242,46.825,158.734
C05997=1026.514,104.872,-104.568,168.239,46.829,158.735
C05998=1026.508,104.623,-104.548,168.237,46.832,158.735
C05999=1026.503,104.374,-104.528,168.234,46.835,158.735
C06000=1026.496,104.125,-104.510,168.231,46.839,158.736
C06001=1026.490,103.875,-104.490,168.229,46.842,158.736
C06002=1026.485,103.626,-104.471,168.226,46.846,158.736
C06003=1026.478,103.377,-104.453,168.224,46.849,158.737
C06004=1026.473,103.127,-104.433,168.221,46.852,158.737
C06005=1026.467,102.878,-104.414,168.218,46.856,158.737
C06006=1026.461,102.629,-104.395,168.216,46.859,158.738
C06007=1026.455,102.381,-104.376,168.213,46.862,158.738
C06008=1026.449,102.131,-104.357,168.211,46.866,158.738
C06009=1026.443,101.882,-104.338,168.208,46.869,158.739
C06010=1026.437,101.633,-104.319,168.206,46.872,158.739
C06011=1026.432,101.383,-104.299,168.203,46.876,158.739
C06012=1026.425,101.134,-104.281,168.200,46.879,158.739
C06013=1026.420,100.885,-104.262,168.198,46.882,158.740
C06014=1026.414,100.636,-104.243,168.195,46.886,158.740
C06015=1026.408,100.387,-104.224,168.193,46.889,158.741
C06016=1026.402,100.138,-104.205,168.190,46.893,158.741
C06017=1026.397,99.888,-104.186,168.188,46.896,158.741
C06018=1026.390,99.639,-104.167,168.185,46.899,158.742
C06019=1026.385,99.390,-104.148,168.182,46.903,158.742
C06020=1026.378,99.140,-104.129,168.180,46.906,158.742
C06021=1026.372,98.891,-104.110,168.177,46.910,158.743
C06022=1026.366,98.641,-104.092,168.175,46.913,158.743
C06023=1026.361,98.393,-104.074,168.172,46.917,158.743
C06024=1026.355,98.143,-104.054,168.169,46.920,158.744
C06025=1026.348,97.894,-104.036,168.167,46.924,158.744
C06026=1026.342,97.645,-104.017,168.164,46.927,158.744
C06027=1026.336,97.396,-103.998,168.161,46.931,158.745
C06028=1026.330,97.147,-103.979,168.159,46.934,158.745
C06029=1026.325,96.897,-103.961,168.156,46.937,158.745
C06030=1026.319,96.648,-103.942,168.154,46.941,158.746
C06031=1026.312,96.399,-103.924,168.151,46.944,158.746
C06032=1026.307,96.150,-103.904,168.148,46.948,158.746
C06033=1026.300,95.900,-103.886,168.146,46.951,158.747
C06034=1026.294,95.651,-103.867,168.143,46.955,158.747
C06035=1026.289,95.402,-103.849,168.141,46.958,158.748
C06036=1026.282,95.153,-103.830,168.138,46.962,158.748
C06037=1026.277,94.903,-103.811,168.135,46.965,158.748
C06038=1026.270,94.654,-103.792,168.133,46.968,158.749
C06039=1026.264,94.405,-103.774,168.130,46.972,158.749
C06040=1026.259,94.156,-103.756,168.128,46.975,158.749
C06041=1026.253,93.907,-103.737,168.125,46.979,158.750
C06042=1026.247,93.657,-103.718,168.123,46.982,158.750
C06043=1026.241,93.408,-103.700,168.120,46.985,158.750
C06044=1026.235,93.159,-103.681,168.117,46.989,158.750
C06045=1026.229,92.910,-103.662,168.115,46.992,158.751
C06046=1026.223,92.661,-103.644,168.112,46.996,158.751
C06047=1026.217,92.411,-103.626,168.110,46.999,158.752
C06048=1026.211,92.127,-103.604,168.107,47.003,158.752
C06049=1026.204,91.843,-103.583,168.105,47.007,158.752
C06050=1026.197,91.557,-103.562,168.102,47.011,158.753
C06051=1026.190,91.273,-103.541,168.099,47.014,158.753
C06052=1026.184,91.024,-103.522,168.096,47.018,158.754
C06053=1026.179,90.775,-103.503,168.093,47.021,158.754
C06054=1026.172,90.525,-103.485,168.091,47.025,158.754
C06055=1026.167,90.276,-103.466,168.088,47.028,158.755
C06056=1026.161,90.026,-103.448,168.086,47.031,158.755
C06057=1026.155,89.778,-103.430,168.083,47.035,158.755
C06058=1026.149,89.528,-103.411,168.081,47.039,158.756
C06059=1026.143,89.279,-103.393,168.078,47.042,158.756
C06060=1026.137,89.030,-103.374,168.075,47.045,158.756
C06061=1026.131,88.781,-103.356,168.073,47.049,158.757
C06062=1026.125,88.531,-103.338,168.070,47.053,158.757
C06063=1026.119,88.282,-103.320,168.068,47.056,158.757
C06064=1026.113,88.033,-103.302,168.065,47.059,158.758
C06065=1026.107,87.783,-103.284,168.062,47.063,158.758
C06066=1026.100,87.534,-103.265,168.060,47.066,158.758
C06067=1026.094,87.285,-103.247,168.057,47.070,158.759
C06068=1026.089,87.036,-103.228,168.055,47.074,158.759
C06069=1026.083,86.786,-103.210,168.052,47.077,158.759
C06070=1026.076,86.537,-103.192,168.049,47.080,158.760
C06071=1026.071,86.288,-103.174,168.047,47.084,158.760
C06072=1026.064,86.039,-103.155,168.045,47.088,158.760
C06073=1026.058,85.789,-103.137,168.042,47.090,158.761
C06074=1026.053,85.540,-103.120,168.039,47.094,158.761
C06075=1026.046,85.291,-103.101,168.037,47.098,158.761
C06076=1026.040,85.041,-103.083,168.035,47.101,158.762
C06077=1026.034,84.793,-103.065,168.031,47.104,158.762
C06078=1026.028,84.543,-103.047,168.030,47.108,158.762
C06079=1026.022,84.293,-103.029,168.027,47.112,158.763
C06080=1026.016,84.045,-103.011,168.025,47.115,158.763
C06081=1026.010,83.795,-102.993,168.022,47.118,158.763
C06082=1026.004,83.546,-102.974,168.019,47.122,158.764
C06083=1025.998,83.297,-102.957,168.017,47.125,158.764
C06084=1025.992,83.047,-102.939,168.014,47.129,158.765
C06085=1025.987,82.798,-102.920,168.012,47.132,158.765
C06086=1025.981,82.549,-102.902,168.009,47.136,158.765
C06087=1025.975,82.299,-102.884,168.007,47.139,158.766
C06088=1025.969,82.051,-102.866,168.004,47.143,158.766
C06089=1025.963,81.801,-102.848,168.001,47.146,158.766
C06090=1025.957,81.551,-102.830,167.999,47.150,158.767
C06091=1025.951,81.303,-102.812,167.996,47.153,158.767
C06092=1025.945,81.053,-102.794,167.994,47.156,158.767
C06093=1025.939,80.804,-102.776,167.991,47.160,158.768
C06094=1025.933,80.555,-102.757,167.989,47.163,158.768
C06095=1025.927,80.305,-102.740,167.986,47.166,158.768
C06096=1025.921,80.056,-102.722,167.984,47.170,158.769
C06097=1025.915,79.807,-102.703,167.981,47.174,158.769
C06098=1025.909,79.558,-102.686,167.978,47.178,158.769
C06099=1025.903,79.308,-102.668,167.976,47.180,158.770
C06100=1025.898,79.059,-102.650,167.973,47.184,158.770
C06101=1025.891,78.810,-102.632,167.971,47.188,158.770
C06102=1025.885,78.560,-102.614,167.968,47.191,158.771
C06103=1025.880,78.311,-102.596,167.966,47.194,158.771
C06104=1025.874,78.061,-102.578,167.963,47.198,158.771
C06105=1025.868,77.813,-102.560,167.961,47.201,158.772
C06106=1025.862,77.563,-102.542,167.958,47.204,158.772
C06107=1025.856,77.314,-102.524,167.956,47.208,158.772
C06108=1025.850,77.064,-102.506,167.953,47.211,158.773
C06109=1025.844,76.815,-102.489,167.950,47.215,158.773
C06110=1025.838,76.566,-102.471,167.948,47.218,158.773
C06111=1025.832,76.316,-102.453,167.946,47.222,158.774
C06112=1025.825,76.032,-102.433,167.943,47.226,158.774
C06113=1025.818,75.747,-102.413,167.940,47.230,158.774
C06114=1025.811,75.463,-102.393,167.937,47.234,158.775
C06115=1025.805,75.178,-102.372,167.934,47.238,158.775
C06116=1025.799,74.929,-102.355,167.931,47.242,158.776
C06117=1025.792,74.679,-102.338,167.929,47.244,158.776
C06118=1025.787,74.430,-102.320,167.926,47.248,158.776
C06119=1025.780,74.181,-102.301,167.924,47.252,158.777
C06120=1025.775,73.932,-102.284,167.922,47.255,158.777
C06121=1025.768,73.683,-102.266,167.919,47.259,158.777
C06122=1025.763,73.434,-102.249,167.917,47.262,158.778
C06123=1025.756,73.184,-102.231,167.914,47.266,158.778
C06124=1025.751,72.935,-102.213,167.912,47.269,158.779
C06125=1025.744,72.686,-102.196,167.909,47.273,158.779
C06126=1025.739,72.437,-102.178,167.907,47.276,158.779
C06127=1025.732,72.187,-102.160,167.904,47.280,158.779
C06128=1025.727,71.938,-102.143,167.902,47.283,158.780
C06129=1025.720,71.688,-102.126,167.899,47.287,158.780
C06130=1025.715,71.439,-102.108,167.896,47.290,158.780
C06131=1025.709,71.189,-102.091,167.894,47.294,158.781
C06132=1025.703,70.940,-102.073,167.891,47.297,158.781
C06133=1025.696,70.690,-102.056,167.889,47.300,158.781
C06134=1025.691,70.441,-102.038,167.886,47.304,158.782
C06135=1025.685,70.192,-102.020,167.884,47.307,158.782
C06136=1025.678,69.943,-102.003,167.881,47.311,158.783
C06137=1025.673,69.694,-101.986,167.878,47.314,158.783
C06138=1025.667,69.444,-101.968,167.876,47.318,158.783
C06139=1025.661,69.195,-101.951,167.873,47.322,158.784
C06140=1025.654,68.946,-101.933,167.871,47.325,158.784
C06141=1025.649,68.697,-101.915,167.868,47.328,158.784
C06142=1025.642,68.447,-101.899,167.866,47.332,158.785
C06143=1025.637,68.198,-101.881,167.864,47.335,158.785
C06144=1025.631,67.948,-101.863,167.862,47.339,158.785
C06145=1025.624,67.699,-101.846,167.858,47.342,158.786
C06146=1025.619,67.450,-101.829,167.856,47.346,158.786
C06147=1025.612,67.200,-101.812,167.854,47.349,158.786
C06148=1025.607,66.951,-101.795,167.851,47.353,158.787
C06149=1025.600,66.702,-101.777,167.849,47.356,158.787
C06150=1025.594,66.452,-101.760,167.846,47.360,158.787
C06151=1025.589,66.203,-101.742,167.843,47.364,158.788
C06152=1025.582,65.953,-101.726,167.841,47.367,158.788
C06153=1025.577,65.704,-101.708,167.838,47.370,158.788
C06154=1025.570,65.455,-101.691,167.836,47.374,158.789
C06155=1025.565,65.205,-101.674,167.833,47.377,158.789
C06156=1025.559,64.957,-101.657,167.831,47.381,158.789
C06157=1025.552,64.707,-101.639,167.828,47.385,158.790
C06158=1025.546,64.458,-101.622,167.825,47.388,158.790
C06159=1025.540,64.208,-101.605,167.823,47.391,158.790
C06160=1025.534,63.959,-101.588,167.820,47.395,158.791
C06161=1025.529,63.710,-101.570,167.819,47.399,158.791
C06162=1025.522,63.460,-101.553,167.815,47.402,158.791
C06163=1025.517,63.211,-101.536,167.814,47.405,158.792
C06164=1025.510,62.961,-101.519,167.811,47.409,158.792
C06165=1025.504,62.712,-101.502,167.808,47.413,158.793
C06166=1025.498,62.463,-101.485,167.806,47.416,158.793
C06167=1025.492,62.213,-101.468,167.803,47.420,158.793
C06168=1025.485,61.964,-101.451,167.800,47.424,158.794
C06169=1025.479,61.715,-101.435,167.798,47.427,158.794
C06170=1025.473,61.465,-101.418,167.795,47.431,158.794
C06171=1025.467,61.216,-101.401,167.792,47.434,158.795
C06172=1025.461,60.966,-101.383,167.790,47.438,158.795
C06173=1025.455,60.717,-101.367,167.787,47.442,158.795
C06174=1025.448,60.468,-101.350,167.785,47.445,158.796
C06175=1025.442,60.218,-101.333,167.783,47.449,158.796
C06176=1025.436,59.977,-101.317,167.780,47.453,158.796
C06177=1025.430,59.735,-101.300,167.778,47.456,158.797
C06178=1025.425,59.492,-101.284,167.775,47.459,158.797
C06179=1025.419,59.251,-101.268,167.773,47.463,158.798
C06180=1025.413,59.009,-101.252,167.770,47.467,158.798
C06181=1025.407,58.767,-101.235,167.768,47.470,158.798
C06182=1025.401,58.526,-101.220,167.765,47.473,158.798
C06183=1025.395,58.284,-101.203,167.763,47.477,158.799
C06184=1025.389,58.035,-101.186,167.760,47.481,158.799
C06185=1025.382,57.785,-101.169,167.757,47.484,158.800
C06186=1025.377,57.535,-101.152,167.755,47.487,158.800
C06187=1025.371,57.286,-101.135,167.752,47.491,158.800
C06188=1025.364,57.036,-101.119,167.751,47.495,158.801
C06189=1025.358,56.788,-101.102,167.748,47.498,158.801
C06190=1025.352,56.538,-101.086,167.745,47.502,158.801
C06191=1025.347,56.289,-101.069,167.743,47.505,158.802
C06192=1025.340,56.039,-101.051,167.740,47.509,158.802
C06193=1025.334,55.790,-101.035,167.738,47.512,158.802
C06194=1025.328,55.541,-101.018,167.735,47.516,158.803
C06195=1025.321,55.291,-101.001,167.732,47.520,158.803
C06196=1025.316,55.041,-100.985,167.730,47.523,158.803
C06197=1025.310,54.793,-100.968,167.727,47.527,158.804
C06198=1025.304,54.543,-100.951,167.725,47.530,158.804
C06199=1025.298,54.294,-100.935,167.722,47.534,158.804
C06200=1025.291,54.045,-100.918,167.719,47.538,158.805
C06201=1025.286,53.795,-100.901,167.717,47.541,158.805
C06202=1025.280,53.546,-100.885,167.714,47.544,158.805
C06203=1025.273,53.297,-100.868,167.713,47.548,158.806
C06204=1025.267,53.047,-100.851,167.710,47.552,158.806
C06205=1025.261,52.797,-100.835,167.707,47.555,158.806
C06206=1025.255,52.548,-100.819,167.705,47.558,158.807
C06207=1025.249,52.299,-100.801,167.702,47.562,158.807
C06208=1025.242,51.999,-100.781,167.699,47.566,158.807
C06209=1025.235,51.700,-100.761,167.696,47.571,158.808
C06210=1025.227,51.400,-100.742,167.692,47.575,158.808
C06211=1025.220,51.100,-100.722,167.690,47.579,158.809
C06212=1025.215,50.851,-100.704,167.687,47.583,158.809
C06213=1025.208,50.601,-100.688,167.685,47.586,158.809
C06214=1025.202,50.351,-100.672,167.682,47.590,158.810
C06215=1025.196,50.102,-100.655,167.680,47.593,158.810
C06216=1025.190,49.853,-100.638,167.677,47.597,158.810
C06217=1025.184,49.604,-100.622,167.674,47.600,158.811
C06218=1025.179,49.354,-100.605,167.672,47.604,158.811
C06219=1025.172,49.104,-100.589,167.669,47.607,158.811
C06220=1025.166,48.855,-100.572,167.667,47.610,158.812
C06221=1025.160,48.606,-100.555,167.664,47.614,158.812
C06222=1025.154,48.357,-100.539,167.663,47.618,158.812
C06223=1025.149,48.107,-100.522,167.659,47.621,158.813
C06224=1025.143,47.858,-100.506,167.656,47.625,158.813
C06225=1025.137,47.608,-100.490,167.655,47.628,158.813
C06226=1025.131,47.359,-100.474,167.651,47.631,158.813
C06227=1025.124,47.110,-100.456,167.650,47.635,158.814
C06228=1025.118,46.860,-100.440,167.647,47.639,158.814
C06229=1025.113,46.611,-100.423,167.645,47.641,158.814
C06230=1025.107,46.361,-100.407,167.642,47.645,158.815
C06231=1025.101,46.112,-100.391,167.640,47.649,158.815
C06232=1025.095,45.863,-100.374,167.637,47.652,158.815
C06233=1025.089,45.613,-100.358,167.634,47.656,158.816
C06234=1025.083,45.365,-100.341,167.632,47.659,158.816
C06235=1025.077,45.115,-100.325,167.629,47.662,158.816
C06236=1025.072,44.866,-100.308,167.627,47.666,158.817
C06237=1025.066,44.616,-100.292,167.624,47.669,158.817
C06238=1025.060,44.367,-100.275,167.622,47.673,158.817
C06239=1025.054,44.118,-100.259,167.619,47.676,158.818
C06240=1025.047,43.833,-100.240,167.616,47.680,158.818
C06241=1025.040,43.547,-100.222,167.613,47.684,158.818
C06242=1025.034,43.262,-100.202,167.611,47.688,158.819
C06243=1025.027,42.976,-100.184,167.608,47.692,158.819
C06244=1025.021,42.727,-100.168,167.605,47.695,158.819
C06245=1025.015,42.478,-100.152,167.603,47.698,158.820
C06246=1025.009,42.228,-100.135,167.600,47.702,158.820
C06247=1025.003,41.979,-100.119,167.598,47.706,158.820
C06248=1024.997,41.730,-100.103,167.595,47.710,158.821
C06249=1024.990,41.481,-100.087,167.592,47.713,158.821
C06250=1024.984,41.231,-100.071,167.590,47.716,158.821
C06251=1024.979,40.982,-100.055,167.587,47.720,158.822
C06252=1024.973,40.733,-100.038,167.585,47.724,158.822
C06253=1024.967,40.483,-100.022,167.582,47.727,158.822
C06254=1024.961,40.233,-100.007,167.579,47.731,158.823
C06255=1024.955,39.984,-99.990,167.577,47.734,158.823
C06256=1024.949,39.735,-99.974,167.574,47.737,158.823
C06257=1024.942,39.485,-99.958,167.572,47.741,158.824
C06258=1024.936,39.236,-99.942,167.570,47.745,158.824
C06259=1024.930,38.987,-99.926,167.567,47.748,158.824
C06260=1024.925,38.737,-99.910,167.565,47.751,158.825
C06261=1024.919,38.487,-99.894,167.562,47.755,158.825
C06262=1024.913,38.238,-99.878,167.559,47.759,158.825
C06263=1024.907,37.989,-99.862,167.557,47.762,158.825
C06264=1024.901,37.739,-99.845,167.554,47.766,158.826
C06265=1024.894,37.490,-99.830,167.552,47.769,158.826
C06266=1024.889,37.240,-99.814,167.549,47.772,158.826
C06267=1024.883,36.991,-99.798,167.547,47.776,158.827
C06268=1024.877,36.742,-99.782,167.544,47.780,158.827
C06269=1024.871,36.492,-99.765,167.541,47.784,158.828
C06270=1024.864,36.243,-99.750,167.539,47.786,158.828
C06271=1024.858,35.993,-99.734,167.536,47.790,158.828
C06272=1024.852,35.744,-99.719,167.533,47.794,158.828
C06273=1024.846,35.494,-99.703,167.532,47.798,158.829
C06274=1024.840,35.245,-99.687,167.529,47.802,158.829
C06275=1024.834,34.995,-99.672,167.526,47.805,158.829
C06276=1024.828,34.746,-99.656,167.524,47.808,158.830
C06277=1024.822,34.497,-99.639,167.521,47.812,158.830
C06278=1024.816,34.247,-99.624,167.518,47.816,158.830
C06279=1024.810,33.998,-99.608,167.516,47.819,158.831
C06280=1024.804,33.749,-99.593,167.513,47.823,158.831
C06281=1024.798,33.499,-99.577,167.510,47.826,158.831
C06282=1024.792,33.250,-99.561,167.508,47.830,158.832
C06283=1024.786,33.000,-99.546,167.506,47.834,158.832
C06284=1024.780,32.751,-99.530,167.502,47.837,158.832
C06285=1024.774,32.502,-99.513,167.501,47.841,158.833
C06286=1024.767,32.252,-99.499,167.498,47.844,158.833
C06287=1024.761,32.003,-99.482,167.496,47.847,158.833
C06288=1024.755,31.753,-99.467,167.493,47.851,158.834
C06289=1024.749,31.504,-99.451,167.490,47.855,158.834
C06290=1024.743,31.254,-99.436,167.488,47.858,158.834
C06291=1024.737,31.005,-99.420,167.485,47.862,158.835
C06292=1024.732,30.755,-99.405,167.482,47.865,158.835
C06293=1024.725,30.506,-99.389,167.480,47.869,158.835
C06294=1024.719,30.257,-99.373,167.477,47.873,158.836
C06295=1024.713,30.007,-99.357,167.474,47.876,158.836
C06296=1024.707,29.758,-99.342,167.472,47.880,158.836
C06297=1024.701,29.508,-99.326,167.469,47.883,158.837
C06298=1024.695,29.259,-99.310,167.467,47.886,158.837
C06299=1024.689,29.010,-99.295,167.464,47.890,158.837
C06300=1024.683,28.760,-99.279,167.462,47.894,158.837
C06301=1024.677,28.511,-99.264,167.459,47.897,158.838
C06302=1024.671,28.261,-99.248,167.457,47.901,158.838
C06303=1024.665,28.011,-99.232,167.454,47.905,158.838
C06304=1024.658,27.727,-99.215,167.451,47.908,158.839
C06305=1024.651,27.442,-99.197,167.448,47.912,158.839
C06306=1024.645,27.157,-99.179,167.446,47.917,158.840
C06307=1024.637,26.871,-99.162,167.443,47.921,158.840
C06308=1024.631,26.622,-99.146,167.440,47.924,158.840
C06309=1024.626,26.373,-99.132,167.437,47.928,158.840
C06310=1024.619,26.124,-99.116,167.435,47.931,158.841
C06311=1024.613,25.874,-99.100,167.432,47.935,158.841
C06312=1024.607,25.624,-99.085,167.429,47.939,158.841
C06313=1024.601,25.374,-99.070,167.427,47.942,158.842
C06314=1024.595,25.125,-99.054,167.424,47.946,158.842
C06315=1024.589,24.876,-99.040,167.421,47.950,158.842
C06316=1024.583,24.626,-99.024,167.419,47.953,158.843
C06317=1024.576,24.377,-99.008,167.416,47.956,158.843
C06318=1024.570,24.127,-98.993,167.413,47.960,158.843
C06319=1024.564,23.877,-98.978,167.411,47.964,158.844
C06320=1024.559,23.628,-98.963,167.409,47.968,158.844
C06321=1024.553,23.379,-98.947,167.406,47.971,158.844
C06322=1024.546,23.129,-98.932,167.403,47.975,158.845
C06323=1024.540,22.880,-98.917,167.401,47.978,158.845
C06324=1024.535,22.631,-98.902,167.398,47.982,158.845
C06325=1024.528,22.382,-98.886,167.395,47.985,158.845
C06326=1024.522,22.132,-98.871,167.393,47.989,158.846
C06327=1024.516,21.882,-98.856,167.390,47.993,158.846
C06328=1024.510,21.633,-98.841,167.387,47.996,158.846
C06329=1024.504,21.383,-98.826,167.385,47.999,158.847
C06330=1024.498,21.134,-98.810,167.382,48.003,158.847
C06331=1024.492,20.884,-98.795,167.380,48.007,158.847
C06332=1024.486,20.635,-98.781,167.377,48.010,158.848
C06333=1024.480,20.385,-98.765,167.375,48.014,158.848
C06334=1024.474,20.136,-98.750,167.372,48.018,158.848
C06335=1024.469,19.886,-98.735,167.370,48.021,158.849
C06336=1024.462,19.637,-98.719,167.367,48.024,158.849
C06337=1024.456,19.388,-98.704,167.364,48.028,158.849
C06338=1024.449,19.138,-98.689,167.362,48.031,158.849
C06339=1024.444,18.889,-98.674,167.359,48.035,158.850
C06340=1024.438,18.639,-98.659,167.356,48.039,158.850
C06341=1024.432,18.389,-98.644,167.354,48.042,158.851
C06342=1024.426,18.141,-98.630,167.351,48.046,158.851
C06343=1024.420,17.891,-98.614,167.348,48.049,158.851
C06344=1024.414,17.641,-98.599,167.345,48.053,158.851
C06345=1024.407,17.391,-98.584,167.344,48.057,158.852
C06346=1024.402,17.142,-98.570,167.341,48.060,158.852
C06347=1024.395,16.893,-98.555,167.338,48.064,158.852
C06348=1024.390,16.643,-98.539,167.336,48.068,158.853
C06349=1024.384,16.394,-98.525,167.333,48.071,158.853
C06350=1024.377,16.144,-98.510,167.330,48.075,158.853
C06351=1024.371,15.894,-98.495,167.328,48.078,158.854
C06352=1024.365,15.645,-98.480,167.325,48.082,158.854
C06353=1024.360,15.395,-98.465,167.322,48.085,158.854
C06354=1024.354,15.147,-98.450,167.319,48.089,158.854
C06355=1024.347,14.897,-98.435,167.317,48.093,158.855
C06356=1024.341,14.647,-98.420,167.314,48.096,158.855
C06357=1024.335,14.398,-98.406,167.311,48.100,158.855
C06358=1024.329,14.149,-98.391,167.310,48.103,158.856
C06359=1024.323,13.899,-98.375,167.306,48.106,158.856
C06360=1024.317,13.650,-98.360,167.304,48.110,158.856
C06361=1024.311,13.400,-98.346,167.302,48.114,158.857
C06362=1024.305,13.150,-98.331,167.299,48.118,158.857
C06363=1024.299,12.901,-98.317,167.296,48.121,158.857
C06364=1024.293,12.651,-98.302,167.293,48.125,158.857
C06365=1024.287,12.402,-98.287,167.291,48.128,158.858
C06366=1024.281,12.153,-98.272,167.288,48.132,158.858
C06367=1024.274,11.903,-98.258,167.285,48.136,158.858
C06368=1024.267,11.619,-98.241,167.283,48.140,158.859
C06369=1024.260,11.336,-98.225,167.279,48.144,158.859
C06370=1024.253,11.052,-98.208,167.276,48.149,158.860
C06371=1024.247,10.769,-98.191,167.273,48.153,158.860
C06372=1024.240,10.519,-98.178,167.271,48.156,158.860
C06373=1024.234,10.270,-98.163,167.268,48.160,158.860
C06374=1024.228,10.020,-98.148,167.266,48.163,158.861
C06375=1024.221,9.770,-98.133,167.263,48.167,158.861
C06376=1024.216,9.521,-98.119,167.260,48.171,158.861
C06377=1024.210,9.271,-98.104,167.257,48.175,158.862
C06378=1024.204,9.022,-98.090,167.254,48.179,158.862
C06379=1024.198,8.772,-98.076,167.252,48.182,158.862
C06380=1024.192,8.523,-98.061,167.249,48.186,158.863
C06381=1024.185,8.273,-98.046,167.246,48.189,158.863
C06382=1024.180,8.024,-98.031,167.244,48.193,158.863
C06383=1024.173,7.774,-98.018,167.242,48.196,158.863
C06384=1024.166,7.525,-98.003,167.239,48.200,158.864
C06385=1024.161,7.276,-97.988,167.236,48.204,158.864
C06386=1024.155,7.026,-97.974,167.233,48.208,158.864
C06387=1024.149,6.777,-97.959,167.231,48.211,158.865
C06388=1024.143,6.526,-97.945,167.228,48.215,158.865
C06389=1024.137,6.277,-97.931,167.225,48.218,158.865
C06390=1024.131,6.028,-97.916,167.222,48.222,158.865
C06391=1024.125,5.778,-97.902,167.220,48.225,158.866
C06392=1024.119,5.528,-97.887,167.217,48.229,158.866
C06393=1024.112,5.280,-97.873,167.215,48.233,158.867
C06394=1024.106,5.030,-97.859,167.211,48.236,158.867
C06395=1024.100,4.781,-97.844,167.210,48.240,158.867
C06396=1024.094,4.530,-97.830,167.207,48.244,158.867
C06397=1024.089,4.281,-97.815,167.204,48.247,158.868
C06398=1024.083,4.032,-97.801,167.201,48.251,158.868
C06399=1024.077,3.782,-97.786,167.199,48.254,158.868
C06400=1024.071,3.533,-97.772,167.196,48.258,158.868
C06401=1024.065,3.283,-97.758,167.193,48.261,158.869
C06402=1024.058,3.034,-97.744,167.190,48.265,158.869
C06403=1024.052,2.784,-97.729,167.188,48.268,158.869
C06404=1024.046,2.535,-97.715,167.185,48.272,158.870
C06405=1024.040,2.285,-97.701,167.182,48.276,158.870
C06406=1024.035,2.036,-97.686,167.179,48.279,158.870
C06407=1024.029,1.786,-97.672,167.177,48.283,158.871
C06408=1024.023,1.537,-97.657,167.175,48.287,158.871
C06409=1024.017,1.287,-97.643,167.172,48.290,158.871
C06410=1024.010,1.038,-97.629,167.169,48.294,158.871
C06411=1024.005,0.788,-97.615,167.167,48.297,158.872
C06412=1023.999,0.539,-97.601,167.164,48.301,158.872
C06413=1023.993,0.289,-97.586,167.161,48.305,158.872
C06414=1023.987,0.040,-97.572,167.158,48.308,158.872
C06415=1023.981,-0.210,-97.558,167.156,48.311,158.873
C06416=1023.975,-0.460,-97.544,167.153,48.315,158.873
C06417=1023.970,-0.709,-97.529,167.150,48.318,158.873
C06418=1023.963,-0.959,-97.515,167.148,48.322,158.874
C06419=1023.957,-1.208,-97.501,167.145,48.325,158.874
C06420=1023.952,-1.457,-97.487,167.142,48.329,158.874
C06421=1023.945,-1.708,-97.473,167.139,48.332,158.874
C06422=1023.940,-1.957,-97.458,167.137,48.336,158.875
C06423=1023.934,-2.206,-97.444,167.134,48.339,158.875
C06424=1023.928,-2.456,-97.429,167.131,48.343,158.875
C06425=1023.922,-2.706,-97.416,167.128,48.347,158.875
C06426=1023.916,-2.955,-97.402,167.126,48.350,158.876
C06427=1023.910,-3.204,-97.387,167.124,48.354,158.876
C06428=1023.904,-3.454,-97.373,167.120,48.357,158.876
C06429=1023.898,-3.704,-97.359,167.119,48.361,158.877
C06430=1023.892,-3.953,-97.345,167.115,48.364,158.877
C06431=1023.887,-4.203,-97.331,167.113,48.368,158.877
C06432=1023.880,-4.485,-97.315,167.110,48.372,158.877
C06433=1023.873,-4.766,-97.300,167.106,48.376,158.878
C06434=1023.866,-5.048,-97.285,167.103,48.380,158.878
C06435=1023.859,-5.330,-97.269,167.101,48.384,158.878
C06436=1023.853,-5.579,-97.255,167.098,48.388,158.879
C06437=1023.847,-5.829,-97.241,167.095,48.391,158.879
C06438=1023.841,-6.079,-97.227,167.092,48.395,158.879
C06439=1023.835,-6.328,-97.214,167.089,48.399,158.879
C06440=1023.829,-6.577,-97.199,167.086,48.403,158.880
C06441=1023.822,-6.827,-97.186,167.084,48.406,158.880
C06442=1023.817,-7.077,-97.172,167.081,48.410,158.880
C06443=1023.810,-7.326,-97.159,167.078,48.414,158.881
C06444=1023.804,-7.576,-97.144,167.076,48.418,158.881
C06445=1023.798,-7.826,-97.131,167.072,48.421,158.881
C06446=1023.793,-8.075,-97.117,167.070,48.425,158.881
C06447=1023.786,-8.324,-97.104,167.068,48.428,158.882
C06448=1023.780,-8.575,-97.090,167.065,48.432,158.882
C06449=1023.774,-8.824,-97.076,167.062,48.435,158.882
C06450=1023.768,-9.073,-97.062,167.059,48.439,158.883
C06451=1023.762,-9.322,-97.049,167.056,48.443,158.883
C06452=1023.756,-9.572,-97.034,167.054,48.446,158.883
C06453=1023.750,-9.822,-97.021,167.051,48.450,158.883
C06454=1023.744,-10.071,-97.007,167.049,48.454,158.884
C06455=1023.738,-10.321,-96.994,167.045,48.457,158.884
C06456=1023.733,-10.570,-96.980,167.043,48.461,158.884
C06457=1023.726,-10.820,-96.966,167.040,48.465,158.885
C06458=1023.720,-11.070,-96.953,167.038,48.468,158.885
C06459=1023.714,-11.319,-96.939,167.035,48.472,158.885
C06460=1023.709,-11.569,-96.925,167.032,48.475,158.885
C06461=1023.702,-11.818,-96.912,167.029,48.479,158.886
C06462=1023.696,-12.068,-96.898,167.026,48.483,158.886
C06463=1023.690,-12.317,-96.885,167.023,48.486,158.886
C06464=1023.685,-12.567,-96.871,167.021,48.490,158.886
C06465=1023.679,-12.816,-96.858,167.018,48.494,158.887
C06466=1023.673,-13.066,-96.844,167.015,48.497,158.887
C06467=1023.666,-13.316,-96.830,167.012,48.501,158.887
C06468=1023.661,-13.566,-96.817,167.009,48.504,158.887
C06469=1023.655,-13.815,-96.804,167.007,48.508,158.888
C06470=1023.649,-14.065,-96.790,167.005,48.512,158.888
C06471=1023.643,-14.314,-96.776,167.001,48.515,158.888
C06472=1023.637,-14.563,-96.763,166.999,48.519,158.889
C06473=1023.631,-14.813,-96.749,166.996,48.522,158.889
C06474=1023.625,-15.063,-96.736,166.993,48.526,158.889
C06475=1023.619,-15.312,-96.722,166.991,48.529,158.889
C06476=1023.613,-15.562,-96.709,166.988,48.533,158.890
C06477=1023.608,-15.812,-96.695,166.985,48.537,158.890
C06478=1023.602,-16.061,-96.682,166.982,48.541,158.890
C06479=1023.595,-16.310,-96.669,166.979,48.544,158.890
C06480=1023.589,-16.560,-96.656,166.976,48.548,158.891
C06481=1023.584,-16.810,-96.642,166.973,48.552,158.891
C06482=1023.577,-17.060,-96.629,166.972,48.555,158.891
C06483=1023.571,-17.309,-96.616,166.968,48.558,158.891
C06484=1023.565,-17.558,-96.602,166.966,48.562,158.892
C06485=1023.560,-17.809,-96.589,166.963,48.566,158.892
C06486=1023.553,-18.058,-96.576,166.960,48.570,158.892
C06487=1023.547,-18.307,-96.563,166.957,48.573,158.893
C06488=1023.541,-18.557,-96.550,166.954,48.577,158.893
C06489=1023.535,-18.806,-96.537,166.951,48.581,158.893
C06490=1023.530,-19.056,-96.523,166.948,48.585,158.893
C06491=1023.523,-19.305,-96.510,166.946,48.588,158.894
C06492=1023.517,-19.555,-96.497,166.944,48.592,158.894
C06493=1023.511,-19.805,-96.483,166.940,48.595,158.894
C06494=1023.505,-20.055,-96.471,166.938,48.599,158.894
C06495=1023.499,-20.304,-96.457,166.935,48.603,158.895
C06496=1023.493,-20.584,-96.443,166.932,48.607,158.895
C06497=1023.486,-20.864,-96.428,166.928,48.611,158.895
C06498=1023.479,-21.144,-96.413,166.925,48.615,158.896
C06499=1023.472,-21.424,-96.398,166.923,48.619,158.896
C06500=1023.466,-21.674,-96.385,166.920,48.623,158.896
C06501=1023.460,-21.923,-96.372,166.917,48.626,158.896
C06502=1023.454,-22.173,-96.359,166.914,48.630,158.897
C06503=1023.448,-22.423,-96.346,166.911,48.634,158.897
C06504=1023.443,-22.673,-96.333,166.908,48.637,158.897
C06505=1023.437,-22.922,-96.320,166.905,48.641,158.897
C06506=1023.430,-23.171,-96.306,166.902,48.645,158.898
C06507=1023.425,-23.421,-96.294,166.899,48.648,158.898
C06508=1023.418,-23.670,-96.281,166.897,48.652,158.898
C06509=1023.412,-23.920,-96.268,166.895,48.656,158.899
C06510=1023.407,-24.170,-96.254,166.891,48.659,158.899
C06511=1023.401,-24.420,-96.242,166.889,48.663,158.899
C06512=1023.395,-24.669,-96.228,166.885,48.666,158.899
C06513=1023.389,-24.919,-96.216,166.883,48.670,158.899
C06514=1023.383,-25.168,-96.202,166.880,48.674,158.900
C06515=1023.377,-25.417,-96.190,166.877,48.678,158.900
C06516=1023.372,-25.667,-96.176,166.875,48.681,158.900
C06517=1023.366,-25.917,-96.164,166.872,48.684,158.900
C06518=1023.360,-26.166,-96.151,166.869,48.688,158.901
C06519=1023.354,-26.416,-96.138,166.866,48.692,158.901
C06520=1023.348,-26.665,-96.125,166.863,48.696,158.901
C06521=1023.342,-26.915,-96.112,166.860,48.699,158.901
C06522=1023.337,-27.165,-96.099,166.857,48.703,158.902
C06523=1023.330,-27.415,-96.086,166.854,48.707,158.902
C06524=1023.324,-27.664,-96.073,166.852,48.710,158.902
C06525=1023.318,-27.914,-96.060,166.849,48.714,158.902
C06526=1023.312,-28.164,-96.047,166.847,48.717,158.903
C06527=1023.307,-28.413,-96.035,166.844,48.721,158.903
C06528=1023.300,-28.662,-96.023,166.841,48.725,158.903
C06529=1023.294,-28.912,-96.010,166.838,48.729,158.903
C06530=1023.288,-29.162,-95.997,166.835,48.733,158.904
C06531=1023.282,-29.411,-95.985,166.832,48.736,158.904
C06532=1023.276,-29.661,-95.972,166.829,48.740,158.904
C06533=1023.270,-29.911,-95.959,166.826,48.744,158.905
C06534=1023.264,-30.160,-95.947,166.824,48.748,158.905
C06535=1023.258,-30.410,-95.934,166.820,48.751,158.905
C06536=1023.253,-30.660,-95.922,166.818,48.755,158.905
C06537=1023.247,-30.909,-95.909,166.815,48.759,158.906
C06538=1023.240,-31.158,-95.897,166.812,48.762,158.906
C06539=1023.234,-31.408,-95.884,166.809,48.766,158.906
C06540=1023.228,-31.658,-95.871,166.806,48.770,158.906
C06541=1023.222,-31.907,-95.858,166.803,48.773,158.906
C06542=1023.216,-32.157,-95.846,166.800,48.777,158.907
C06543=1023.211,-32.406,-95.833,166.797,48.781,158.907
C06544=1023.205,-32.656,-95.821,166.794,48.784,158.907
C06545=1023.199,-32.906,-95.808,166.791,48.788,158.907
C06546=1023.193,-33.156,-95.796,166.790,48.792,158.908
C06547=1023.186,-33.405,-95.783,166.787,48.795,158.908
C06548=1023.181,-33.654,-95.771,166.784,48.799,158.908
C06549=1023.175,-33.904,-95.758,166.781,48.803,158.909
C06550=1023.169,-34.154,-95.746,166.778,48.806,158.909
C06551=1023.163,-34.404,-95.733,166.775,48.810,158.909
C06552=1023.157,-34.654,-95.721,166.772,48.813,158.909
C06553=1023.152,-34.903,-95.709,166.769,48.817,158.909
C06554=1023.146,-35.153,-95.696,166.766,48.821,158.910
C06555=1023.140,-35.402,-95.684,166.763,48.825,158.910
C06556=1023.133,-35.652,-95.671,166.760,48.828,158.910
C06557=1023.128,-35.901,-95.659,166.757,48.832,158.910
C06558=1023.122,-36.151,-95.646,166.754,48.836,158.911
C06559=1023.116,-36.401,-95.633,166.752,48.840,158.911
C06560=1023.109,-36.680,-95.620,166.749,48.844,158.911
C06561=1023.103,-36.959,-95.606,166.745,48.848,158.911
C06562=1023.097,-37.238,-95.592,166.742,48.852,158.912
C06563=1023.090,-37.517,-95.578,166.739,48.856,158.912
C06564=1023.084,-37.767,-95.566,166.736,48.859,158.912
C06565=1023.079,-38.016,-95.553,166.733,48.863,158.912
C06566=1023.073,-38.266,-95.541,166.730,48.866,158.913
C06567=1023.067,-38.515,-95.529,166.728,48.870,158.913
C06568=1023.061,-38.765,-95.516,166.724,48.873,158.913
C06569=1023.055,-39.015,-95.504,166.722,48.877,158.913
C06570=1023.049,-39.265,-95.492,166.719,48.881,158.914
C06571=1023.044,-39.515,-95.480,166.716,48.885,158.914
C06572=1023.037,-39.764,-95.468,166.713,48.889,158.914
C06573=1023.031,-40.014,-95.456,166.710,48.892,158.914
C06574=1023.026,-40.263,-95.443,166.707,48.896,158.915
C06575=1023.019,-40.513,-95.431,166.704,48.900,158.915
C06576=1023.013,-40.763,-95.419,166.701,48.904,158.915
C06577=1023.008,-41.012,-95.408,166.699,48.908,158.915
C06578=1023.002,-41.262,-95.395,166.696,48.911,158.915
C06579=1022.996,-41.512,-95.383,166.693,48.915,158.916
C06580=1022.990,-41.761,-95.371,166.690,48.919,158.916
C06581=1022.984,-42.011,-95.359,166.687,48.922,158.916
C06582=1022.978,-42.261,-95.347,166.684,48.926,158.916
C06583=1022.972,-42.510,-95.335,166.681,48.930,158.917
C06584=1022.966,-42.760,-95.323,166.678,48.934,158.917
C06585=1022.960,-43.010,-95.311,166.675,48.937,158.917
C06586=1022.954,-43.259,-95.299,166.673,48.941,158.917
C06587=1022.948,-43.509,-95.287,166.670,48.945,158.918
C06588=1022.943,-43.758,-95.275,166.667,48.948,158.918
C06589=1022.937,-44.008,-95.263,166.664,48.952,158.918
C06590=1022.931,-44.258,-95.251,166.661,48.956,158.918
C06591=1022.925,-44.507,-95.239,166.658,48.960,158.919
C06592=1022.919,-44.757,-95.227,166.655,48.964,158.919
C06593=1022.913,-45.006,-95.215,166.652,48.967,158.919
C06594=1022.907,-45.256,-95.204,166.649,48.971,158.919
C06595=1022.901,-45.506,-95.191,166.646,48.975,158.920
C06596=1022.896,-45.755,-95.179,166.643,48.978,158.920
C06597=1022.889,-46.006,-95.168,166.641,48.982,158.920
C06598=1022.884,-46.255,-95.156,166.638,48.986,158.920
C06599=1022.877,-46.504,-95.144,166.635,48.989,158.920
C06600=1022.872,-46.754,-95.132,166.632,48.993,158.921
C06601=1022.866,-47.004,-95.120,166.629,48.996,158.921
C06602=1022.860,-47.253,-95.108,166.626,49.000,158.921
C06603=1022.855,-47.503,-95.096,166.623,49.004,158.921
C06604=1022.849,-47.752,-95.085,166.620,49.008,158.922
C06605=1022.843,-48.003,-95.073,166.617,49.012,158.922
C06606=1022.837,-48.252,-95.061,166.614,49.015,158.922
C06607=1022.831,-48.502,-95.049,166.611,49.019,158.922
C06608=1022.826,-48.751,-95.038,166.608,49.022,158.922
C06609=1022.820,-49.001,-95.025,166.605,49.026,158.923
C06610=1022.815,-49.251,-95.014,166.603,49.030,158.923
C06611=1022.808,-49.500,-95.002,166.599,49.033,158.923
C06612=1022.803,-49.750,-94.990,166.597,49.037,158.923
C06613=1022.796,-50.000,-94.978,166.594,49.041,158.924
C06614=1022.791,-50.249,-94.967,166.591,49.045,158.924
C06615=1022.785,-50.499,-94.955,166.588,49.048,158.924
C06616=1022.780,-50.749,-94.943,166.585,49.052,158.924
C06617=1022.773,-50.998,-94.931,166.582,49.056,158.925
C06618=1022.767,-51.248,-94.921,166.579,49.059,158.925
C06619=1022.761,-51.498,-94.908,166.576,49.063,158.925
C06620=1022.756,-51.747,-94.897,166.572,49.067,158.925
C06621=1022.749,-51.997,-94.886,166.570,49.071,158.925
C06622=1022.743,-52.246,-94.874,166.567,49.075,158.926
C06623=1022.737,-52.496,-94.863,166.564,49.079,158.926
C06624=1022.731,-52.775,-94.850,166.560,49.083,158.926
C06625=1022.724,-53.056,-94.838,166.557,49.087,158.926
C06626=1022.718,-53.335,-94.825,166.554,49.092,158.927
C06627=1022.711,-53.614,-94.812,166.551,49.096,158.927
C06628=1022.704,-53.865,-94.801,166.547,49.100,158.927
C06629=1022.699,-54.114,-94.790,166.544,49.104,158.927
C06630=1022.693,-54.363,-94.778,166.541,49.108,158.928
C06631=1022.687,-54.613,-94.767,166.539,49.112,158.928
C06632=1022.681,-54.863,-94.756,166.536,49.115,158.928
C06633=1022.675,-55.113,-94.744,166.533,49.119,158.928
C06634=1022.669,-55.362,-94.733,166.530,49.123,158.929
C06635=1022.663,-55.612,-94.722,166.527,49.127,158.929
C06636=1022.657,-55.862,-94.711,166.524,49.130,158.929
C06637=1022.652,-56.112,-94.699,166.520,49.135,158.929
C06638=1022.646,-56.361,-94.688,166.518,49.139,158.930
C06639=1022.639,-56.611,-94.676,166.515,49.143,158.930
C06640=1022.634,-56.860,-94.666,166.512,49.146,158.930
C06641=1022.627,-57.110,-94.654,166.509,49.150,158.930
C06642=1022.622,-57.360,-94.643,166.506,49.154,158.931
C06643=1022.616,-57.609,-94.633,166.503,49.158,158.931
C06644=1022.610,-57.860,-94.621,166.500,49.161,158.931
C06645=1022.604,-58.109,-94.609,166.497,49.165,158.931
C06646=1022.599,-58.358,-94.598,166.494,49.169,158.931
C06647=1022.592,-58.608,-94.587,166.491,49.173,158.932
C06648=1022.586,-58.858,-94.576,166.488,49.177,158.932
C06649=1022.581,-59.107,-94.565,166.485,49.181,158.932
C06650=1022.576,-59.357,-94.554,166.482,49.185,158.932
C06651=1022.569,-59.607,-94.543,166.479,49.188,158.933
C06652=1022.564,-59.857,-94.532,166.476,49.192,158.933
C06653=1022.558,-60.106,-94.521,166.474,49.196,158.933
C06654=1022.552,-60.356,-94.510,166.470,49.199,158.933
C06655=1022.546,-60.605,-94.498,166.468,49.203,158.934
C06656=1022.540,-60.855,-94.487,166.464,49.208,158.934
C06657=1022.534,-61.104,-94.476,166.461,49.211,158.934
///RCONF 1,0,0,1,0,0,0,0,0,0,0,0,0,0,0,0,0,0,0,0,0,0,0,0
C06658=1022.528,-61.355,-94.464,166.458,49.215,158.934
C06659=1022.523,-61.604,-94.453,166.455,49.219,158.934
C06660=1022.517,-61.854,-94.443,166.452,49.222,158.934
C06661=1022.511,-62.103,-94.432,166.449,49.226,158.935
C06662=1022.505,-62.353,-94.420,166.446,49.230,158.935
C06663=1022.499,-62.603,-94.410,166.443,49.233,158.935
C06664=1022.493,-62.852,-94.399,166.441,49.237,158.935
C06665=1022.488,-63.102,-94.388,166.438,49.241,158.936
C06666=1022.483,-63.352,-94.376,166.435,49.245,158.936
C06667=1022.476,-63.602,-94.365,166.431,49.249,158.936
C06668=1022.471,-63.851,-94.354,166.428,49.252,158.936
C06669=1022.465,-64.101,-94.343,166.425,49.256,158.936
C06670=1022.459,-64.350,-94.332,166.422,49.260,158.937
C06671=1022.454,-64.600,-94.322,166.419,49.264,158.937
C06672=1022.447,-64.851,-94.311,166.416,49.268,158.937
C06673=1022.442,-65.100,-94.300,166.413,49.271,158.937
C06674=1022.437,-65.350,-94.289,166.410,49.275,158.937
C06675=1022.431,-65.599,-94.278,166.408,49.279,158.938
C06676=1022.425,-65.849,-94.267,166.405,49.282,158.938
C06677=1022.419,-66.098,-94.256,166.402,49.286,158.938
C06678=1022.414,-66.348,-94.245,166.399,49.289,158.938
C06679=1022.407,-66.598,-94.234,166.395,49.294,158.938
C06680=1022.402,-66.848,-94.223,166.392,49.298,158.939
C06681=1022.396,-67.098,-94.213,166.389,49.301,158.939
C06682=1022.390,-67.347,-94.202,166.386,49.305,158.939
C06683=1022.385,-67.597,-94.191,166.383,49.308,158.939
C06684=1022.380,-67.847,-94.180,166.380,49.312,158.940
C06685=1022.374,-68.096,-94.169,166.377,49.316,158.940
C06686=1022.368,-68.345,-94.158,166.375,49.320,158.940
C06687=1022.363,-68.596,-94.148,166.371,49.323,158.940
C06688=1022.356,-68.876,-94.135,166.368,49.327,158.940
C06689=1022.349,-69.158,-94.123,166.365,49.331,158.940
C06690=1022.343,-69.438,-94.111,166.361,49.336,158.941
C06691=1022.337,-69.719,-94.099,166.358,49.340,158.941
C06692=1022.331,-69.969,-94.088,166.355,49.344,158.941
C06693=1022.326,-70.218,-94.077,166.351,49.347,158.941
C06694=1022.320,-70.468,-94.066,166.349,49.351,158.941
C06695=1022.314,-70.718,-94.056,166.345,49.355,158.942
C06696=1022.309,-70.967,-94.045,166.343,49.359,158.942
C06697=1022.303,-71.217,-94.034,166.340,49.363,158.942
C06698=1022.297,-71.466,-94.023,166.337,49.366,158.942
C06699=1022.292,-71.716,-94.013,166.334,49.370,158.943
C06700=1022.286,-71.966,-94.002,166.331,49.373,158.943
C06701=1022.280,-72.215,-93.991,166.328,49.377,158.943
C06702=1022.275,-72.465,-93.981,166.325,49.380,158.943
C06703=1022.269,-72.715,-93.970,166.322,49.384,158.943
C06704=1022.264,-72.965,-93.959,166.319,49.388,158.943
C06705=1022.259,-73.215,-93.949,166.316,49.391,158.944
C06706=1022.253,-73.464,-93.938,166.313,49.395,158.944
C06707=1022.247,-73.714,-93.927,166.310,49.398,158.944
C06708=1022.242,-73.964,-93.917,166.307,49.402,158.944
C06709=1022.236,-74.213,-93.906,166.304,49.406,158.944
C06710=1022.231,-74.463,-93.896,166.302,49.410,158.945
C06711=1022.225,-74.713,-93.885,166.298,49.414,158.945
C06712=1022.219,-74.963,-93.875,166.295,49.417,158.945
C06713=1022.213,-75.212,-93.864,166.292,49.421,158.945
C06714=1022.208,-75.462,-93.854,166.289,49.425,158.945
C06715=1022.202,-75.712,-93.843,166.286,49.429,158.945
C06716=1022.196,-75.962,-93.833,166.283,49.433,158.946
C06717=1022.190,-76.211,-93.823,166.279,49.437,158.946
C06718=1022.185,-76.461,-93.813,166.276,49.440,158.946
C06719=1022.179,-76.710,-93.802,166.274,49.444,158.946
C06720=1022.174,-76.960,-93.792,166.271,49.448,158.946
C06721=1022.168,-77.210,-93.783,166.268,49.452,158.947
C06722=1022.162,-77.459,-93.772,166.265,49.456,158.947
C06723=1022.157,-77.710,-93.761,166.262,49.459,158.947
C06724=1022.151,-77.959,-93.751,166.259,49.463,158.947
C06725=1022.145,-78.209,-93.740,166.255,49.467,158.948
C06726=1022.139,-78.459,-93.731,166.252,49.471,158.948
C06727=1022.133,-78.708,-93.720,166.249,49.475,158.948
C06728=1022.129,-78.958,-93.710,166.246,49.478,158.948
C06729=1022.123,-79.207,-93.699,166.244,49.482,158.948
C06730=1022.117,-79.457,-93.690,166.241,49.486,158.949
C06731=1022.111,-79.707,-93.680,166.238,49.489,158.949
C06732=1022.106,-79.957,-93.669,166.234,49.494,158.949
C06733=1022.100,-80.207,-93.659,166.231,49.498,158.949
C06734=1022.094,-80.457,-93.649,166.228,49.501,158.949
C06735=1022.089,-80.707,-93.639,166.225,49.505,158.949
C06736=1022.083,-80.956,-93.630,166.223,49.509,158.950
C06737=1022.077,-81.205,-93.619,166.219,49.513,158.950
C06738=1022.071,-81.455,-93.609,166.216,49.517,158.950
C06739=1022.066,-81.705,-93.599,166.213,49.521,158.950
C06740=1022.059,-81.955,-93.589,166.210,49.525,158.951
C06741=1022.054,-82.205,-93.579,166.207,49.529,158.951
C06742=1022.048,-82.454,-93.570,166.204,49.533,158.951
C06743=1022.043,-82.704,-93.559,166.200,49.537,158.951
C06744=1022.037,-82.953,-93.550,166.198,49.541,158.951
C06745=1022.031,-83.204,-93.540,166.195,49.545,158.952
C06746=1022.025,-83.453,-93.530,166.192,49.549,158.952
C06747=1022.020,-83.703,-93.520,166.188,49.552,158.952
C06748=1022.014,-83.953,-93.511,166.185,49.556,158.952
C06749=1022.008,-84.203,-93.500,166.183,49.560,158.952
C06750=1022.002,-84.453,-93.491,166.179,49.564,158.953
C06751=1021.997,-84.703,-93.481,166.176,49.568,158.953
C06752=1021.990,-84.985,-93.469,166.173,49.572,158.953
C06753=1021.984,-85.268,-93.459,166.169,49.577,158.953
C06754=1021.977,-85.550,-93.447,166.166,49.581,158.953
C06755=1021.971,-85.833,-93.437,166.162,49.586,158.954
C06756=1021.966,-86.083,-93.427,166.159,49.590,158.954
C06757=1021.960,-86.333,-93.417,166.156,49.593,158.954
C06758=1021.955,-86.582,-93.407,166.153,49.597,158.954
C06759=1021.949,-86.832,-93.398,166.151,49.601,158.955
C06760=1021.943,-87.082,-93.388,166.148,49.605,158.955
C06761=1021.937,-87.332,-93.378,166.144,49.609,158.955
C06762=1021.931,-87.581,-93.369,166.141,49.613,158.955
C06763=1021.926,-87.831,-93.359,166.138,49.617,158.955
C06764=1021.920,-88.081,-93.349,166.135,49.620,158.955
C06765=1021.915,-88.330,-93.339,166.132,49.624,158.956
C06766=1021.909,-88.580,-93.330,166.129,49.629,158.956
C06767=1021.903,-88.830,-93.320,166.125,49.632,158.956
C06768=1021.898,-89.079,-93.310,166.123,49.636,158.956
C06769=1021.892,-89.330,-93.300,166.120,49.640,158.957
C06770=1021.886,-89.579,-93.291,166.117,49.643,158.957
C06771=1021.881,-89.829,-93.281,166.113,49.648,158.957
C06772=1021.875,-90.079,-93.271,166.110,49.652,158.957
C06773=1021.870,-90.329,-93.261,166.107,49.655,158.957
C06774=1021.864,-90.578,-93.252,166.104,49.659,158.957
C06775=1021.858,-90.828,-93.242,166.102,49.663,158.958
C06776=1021.853,-91.078,-93.233,166.099,49.666,158.958
C06777=1021.847,-91.327,-93.224,166.095,49.671,158.958
C06778=1021.842,-91.577,-93.214,166.092,49.674,158.958
C06779=1021.836,-91.827,-93.204,166.089,49.678,158.958
C06780=1021.831,-92.077,-93.194,166.086,49.682,158.959
C06781=1021.825,-92.326,-93.185,166.083,49.686,158.959
C06782=1021.820,-92.577,-93.176,166.080,49.690,158.959
C06783=1021.814,-92.826,-93.166,166.077,49.694,158.959
C06784=1021.809,-93.076,-93.156,166.073,49.697,158.959
C06785=1021.803,-93.326,-93.147,166.071,49.701,158.959
C06786=1021.797,-93.575,-93.137,166.068,49.705,158.960
C06787=1021.792,-93.825,-93.128,166.065,49.709,158.960
C06788=1021.787,-94.074,-93.119,166.062,49.713,158.960
C06789=1021.781,-94.325,-93.109,166.058,49.716,158.960
C06790=1021.776,-94.574,-93.099,166.055,49.720,158.960
C06791=1021.770,-94.824,-93.089,166.052,49.724,158.960
C06792=1021.765,-95.073,-93.081,166.049,49.728,158.961
C06793=1021.759,-95.323,-93.071,166.047,49.732,158.961
C06794=1021.754,-95.573,-93.061,166.044,49.735,158.961
C06795=1021.748,-95.823,-93.053,166.041,49.739,158.961
C06796=1021.743,-96.072,-93.043,166.037,49.743,158.961
C06797=1021.737,-96.322,-93.033,166.034,49.747,158.962
C06798=1021.732,-96.572,-93.023,166.031,49.750,158.962
C06799=1021.726,-96.822,-93.015,166.028,49.754,158.962
C06800=1021.721,-97.071,-93.005,166.025,49.758,158.962
C06801=1021.716,-97.322,-92.996,166.022,49.762,158.962
C06802=1021.710,-97.571,-92.987,166.020,49.766,158.962
C06803=1021.705,-97.821,-92.976,166.015,49.769,158.962
C06804=1021.699,-98.071,-92.968,166.013,49.774,158.963
C06805=1021.693,-98.321,-92.958,166.010,49.778,158.963
C06806=1021.688,-98.570,-92.950,166.007,49.781,158.963
C06807=1021.682,-98.820,-92.940,166.004,49.785,158.963
C06808=1021.677,-99.070,-92.931,166.000,49.789,158.963
C06809=1021.671,-99.320,-92.922,165.998,49.793,158.964
C06810=1021.666,-99.570,-92.913,165.994,49.797,158.964
C06811=1021.660,-99.820,-92.904,165.992,49.801,158.964
C06812=1021.654,-100.069,-92.895,165.988,49.805,158.964
C06813=1021.649,-100.318,-92.886,165.985,49.809,158.964
C06814=1021.643,-100.569,-92.877,165.982,49.813,158.965
C06815=1021.638,-100.818,-92.867,165.979,49.817,158.965
C06816=1021.633,-101.080,-92.858,165.976,49.821,158.965
C06817=1021.627,-101.342,-92.849,165.973,49.825,158.965
C06818=1021.620,-101.603,-92.839,165.970,49.828,158.965
C06819=1021.614,-101.865,-92.830,165.966,49.833,158.966
C06820=1021.610,-102.114,-92.820,165.963,49.837,158.966
C06821=1021.604,-102.365,-92.812,165.960,49.841,158.966
C06822=1021.598,-102.615,-92.803,165.956,49.845,158.966
C06823=1021.593,-102.864,-92.794,165.954,49.849,158.966
C06824=1021.587,-103.114,-92.785,165.951,49.853,158.967
C06825=1021.582,-103.364,-92.777,165.948,49.856,158.967
C06826=1021.576,-103.613,-92.767,165.945,49.860,158.967
C06827=1021.571,-103.864,-92.758,165.941,49.865,158.967
C06828=1021.566,-104.113,-92.749,165.938,49.868,158.967
C06829=1021.560,-104.362,-92.740,165.935,49.872,158.967
C06830=1021.554,-104.613,-92.731,165.933,49.876,158.968
C06831=1021.549,-104.863,-92.723,165.930,49.880,158.968
C06832=1021.543,-105.112,-92.714,165.926,49.884,158.968
C06833=1021.538,-105.362,-92.705,165.923,49.888,158.968
C06834=1021.532,-105.612,-92.696,165.920,49.892,158.968
C06835=1021.527,-105.861,-92.687,165.917,49.895,158.968
C06836=1021.521,-106.111,-92.678,165.915,49.899,158.969
C06837=1021.516,-106.361,-92.669,165.911,49.904,158.969
C06838=1021.511,-106.611,-92.661,165.908,49.907,158.969
C06839=1021.506,-106.860,-92.652,165.905,49.911,158.969
C06840=1021.500,-107.111,-92.643,165.902,49.915,158.969
C06841=1021.494,-107.360,-92.634,165.899,49.919,158.970
C06842=1021.489,-107.610,-92.626,165.895,49.923,158.970
C06843=1021.483,-107.860,-92.617,165.893,49.927,158.970
C06844=1021.478,-108.110,-92.608,165.889,49.930,158.970
C06845=1021.472,-108.359,-92.599,165.887,49.934,158.970
C06846=1021.467,-108.609,-92.591,165.883,49.939,158.970
C06847=1021.462,-108.859,-92.582,165.880,49.943,158.971
C06848=1021.455,-109.109,-92.574,165.877,49.946,158.971
C06849=1021.450,-109.358,-92.565,165.874,49.950,158.971
C06850=1021.445,-109.608,-92.557,165.872,49.954,158.971
C06851=1021.440,-109.858,-92.549,165.868,49.959,158.971
C06852=1021.434,-110.108,-92.540,165.865,49.962,158.972
C06853=1021.428,-110.358,-92.531,165.862,49.966,158.972
C06854=1021.423,-110.608,-92.523,165.859,49.970,158.972
C06855=1021.418,-110.857,-92.514,165.855,49.974,158.972
C06856=1021.413,-111.107,-92.506,165.852,49.978,158.972
C06857=1021.406,-111.357,-92.496,165.850,49.982,158.973
C06858=1021.401,-111.607,-92.488,165.847,49.986,158.973
C06859=1021.396,-111.856,-92.479,165.844,49.990,158.973
C06860=1021.390,-112.106,-92.471,165.840,49.994,158.973
C06861=1021.385,-112.356,-92.463,165.837,49.998,158.973
C06862=1021.379,-112.605,-92.454,165.834,50.001,158.973
C06863=1021.374,-112.855,-92.446,165.832,50.005,158.974
C06864=1021.368,-113.105,-92.437,165.828,50.010,158.974
C06865=1021.363,-113.356,-92.429,165.825,50.013,158.974
C06866=1021.358,-113.605,-92.421,165.822,50.017,158.974
C06867=1021.353,-113.855,-92.412,165.819,50.021,158.974
C06868=1021.347,-114.128,-92.403,165.816,50.026,158.974
C06869=1021.341,-114.400,-92.394,165.813,50.030,158.975
C06870=1021.335,-114.674,-92.384,165.809,50.034,158.975
C06871=1021.329,-114.947,-92.375,165.805,50.039,158.975
C06872=1021.324,-115.197,-92.367,165.803,50.043,158.975
C06873=1021.319,-115.447,-92.359,165.800,50.047,158.975
C06874=1021.313,-115.696,-92.351,165.797,50.050,158.976
C06875=1021.307,-115.946,-92.342,165.793,50.055,158.976
C06876=1021.302,-116.196,-92.334,165.790,50.059,158.976
C06877=1021.297,-116.445,-92.325,165.787,50.062,158.976
C06878=1021.291,-116.695,-92.318,165.784,50.066,158.976
C06879=1021.286,-116.945,-92.310,165.782,50.070,158.977
C06880=1021.279,-117.230,-92.300,165.778,50.075,158.977
C06881=1021.273,-117.515,-92.291,165.774,50.079,158.977
C06882=1021.267,-117.800,-92.281,165.771,50.084,158.977
C06883=1021.261,-118.085,-92.272,165.767,50.089,158.977
C06884=1021.255,-118.334,-92.263,165.764,50.093,158.977
C06885=1021.250,-118.584,-92.256,165.761,50.096,158.978
C06886=1021.245,-118.834,-92.248,165.758,50.100,158.978
C06887=1021.239,-119.084,-92.239,165.755,50.105,158.978
C06888=1021.234,-119.333,-92.231,165.752,50.109,158.978
C06889=1021.228,-119.584,-92.223,165.749,50.112,158.978
C06890=1021.223,-119.833,-92.215,165.746,50.116,158.979
C06891=1021.218,-120.083,-92.206,165.743,50.120,158.979
C06892=1021.212,-120.333,-92.199,165.740,50.125,158.979
C06893=1021.207,-120.583,-92.191,165.737,50.128,158.979
C06894=1021.202,-120.832,-92.182,165.734,50.132,158.979
C06895=1021.196,-121.082,-92.175,165.731,50.136,158.979
C06896=1021.191,-121.331,-92.167,165.727,50.140,158.979
C06897=1021.186,-121.581,-92.158,165.724,50.144,158.980
C06898=1021.181,-121.831,-92.151,165.722,50.148,158.980
C06899=1021.175,-122.081,-92.143,165.719,50.152,158.980
C06900=1021.170,-122.331,-92.135,165.716,50.156,158.980
C06901=1021.165,-122.581,-92.127,165.712,50.160,158.980
C06902=1021.159,-122.830,-92.119,165.709,50.164,158.981
C06903=1021.154,-123.081,-92.111,165.706,50.167,158.981
C06904=1021.149,-123.330,-92.102,165.703,50.171,158.981
C06905=1021.143,-123.580,-92.095,165.701,50.176,158.981
C06906=1021.138,-123.830,-92.087,165.697,50.180,158.981
C06907=1021.133,-124.080,-92.079,165.694,50.183,158.981
C06908=1021.127,-124.329,-92.071,165.691,50.187,158.982
C06909=1021.122,-124.579,-92.064,165.688,50.192,158.982
C06910=1021.116,-124.829,-92.056,165.684,50.195,158.982
C06911=1021.111,-125.079,-92.048,165.682,50.199,158.982
C06912=1021.105,-125.329,-92.040,165.679,50.203,158.982
C06913=1021.100,-125.579,-92.032,165.676,50.208,158.983
C06914=1021.095,-125.829,-92.024,165.672,50.212,158.983
C06915=1021.089,-126.079,-92.017,165.669,50.215,158.983
C06916=1021.085,-126.328,-92.009,165.667,50.220,158.983
C06917=1021.079,-126.578,-92.001,165.664,50.224,158.983
C06918=1021.074,-126.828,-91.994,165.661,50.228,158.984
C06919=1021.068,-127.077,-91.986,165.657,50.231,158.983
C06920=1021.063,-127.328,-91.978,165.654,50.236,158.984
C06921=1021.058,-127.577,-91.970,165.652,50.240,158.984
C06922=1021.053,-127.827,-91.963,165.649,50.244,158.984
C06923=1021.047,-128.077,-91.956,165.645,50.247,158.984
C06924=1021.042,-128.326,-91.947,165.643,50.251,158.984
C06925=1021.038,-128.575,-91.938,165.640,50.254,158.984
C06926=1021.034,-128.825,-91.928,165.637,50.256,158.984
C06927=1021.031,-129.075,-91.919,165.633,50.258,158.984
C06928=1021.028,-129.325,-91.908,165.632,50.260,158.984
C06929=1021.026,-129.574,-91.897,165.629,50.260,158.984
C06930=1021.023,-129.824,-91.885,165.626,50.261,158.983
C06931=1021.022,-130.074,-91.873,165.624,50.261,158.983
C06932=1021.021,-130.324,-91.860,165.621,50.260,158.982
C06933=1021.021,-130.574,-91.846,165.619,50.259,158.982
C06934=1021.020,-130.823,-91.831,165.617,50.257,158.981
C06935=1021.021,-131.073,-91.817,165.615,50.255,158.981
C06936=1021.021,-131.323,-91.802,165.613,50.253,158.980
C06937=1021.023,-131.572,-91.785,165.611,50.250,158.979
C06938=1021.025,-131.822,-91.769,165.609,50.245,158.978
C06939=1021.027,-132.072,-91.752,165.607,50.242,158.977
C06940=1021.030,-132.322,-91.734,165.606,50.236,158.976
C06941=1021.033,-132.571,-91.717,165.604,50.232,158.975
C06942=1021.037,-132.821,-91.697,165.603,50.226,158.973
C06943=1021.040,-133.071,-91.678,165.601,50.220,158.972
C06944=1020.759,-133.097,-92.035,165.556,50.526,159.017
C06945=1020.755,-132.847,-92.054,165.556,50.532,159.018
C06946=1020.752,-132.597,-92.073,165.558,50.538,159.019
C06947=1020.748,-132.348,-92.091,165.560,50.543,159.020
C06948=1020.746,-132.098,-92.109,165.562,50.547,159.021
C06949=1020.743,-131.849,-92.126,165.563,50.552,159.022
C06950=1020.741,-131.598,-92.142,165.565,50.556,159.023
C06951=1020.741,-131.349,-92.158,165.568,50.559,159.024
C06952=1020.739,-131.098,-92.173,165.569,50.561,159.025
C06953=1020.739,-130.849,-92.188,165.571,50.564,159.026
C06954=1020.739,-130.599,-92.203,165.574,50.566,159.026
C06955=1020.740,-130.349,-92.216,165.576,50.566,159.027
C06956=1020.741,-130.100,-92.229,165.578,50.567,159.027
C06957=1020.742,-129.850,-92.241,165.580,50.567,159.028
C06958=1020.744,-129.601,-92.253,165.584,50.567,159.028
C06959=1020.747,-129.350,-92.265,165.585,50.565,159.028
C06960=1020.749,-129.101,-92.276,165.589,50.564,159.029
C06961=1020.753,-128.851,-92.285,165.591,50.562,159.029
C06962=1020.756,-128.601,-92.295,165.593,50.560,159.029
C06963=1020.761,-128.352,-92.304,165.597,50.557,159.029
C06964=1020.766,-128.102,-92.312,165.600,50.554,159.029
C06965=1020.771,-127.853,-92.319,165.603,50.549,159.029
C06966=1020.776,-127.603,-92.327,165.605,50.545,159.028
C06967=1020.782,-127.354,-92.335,165.609,50.541,159.028
C06968=1020.787,-127.103,-92.343,165.612,50.537,159.028
C06969=1020.792,-126.855,-92.350,165.615,50.533,159.028
C06970=1020.797,-126.604,-92.358,165.617,50.529,159.028
C06971=1020.803,-126.354,-92.365,165.621,50.525,159.028
C06972=1020.808,-126.105,-92.374,165.624,50.521,159.027
C06973=1020.813,-125.854,-92.381,165.627,50.517,159.027
C06974=1020.819,-125.606,-92.389,165.631,50.513,159.027
C06975=1020.823,-125.355,-92.397,165.633,50.509,159.027
C06976=1020.829,-125.105,-92.404,165.636,50.504,159.027
C06977=1020.834,-124.855,-92.412,165.639,50.500,159.026
C06978=1020.840,-124.605,-92.420,165.642,50.496,159.026
C06979=1020.845,-124.356,-92.428,165.646,50.492,159.026
C06980=1020.851,-124.106,-92.435,165.648,50.488,159.026
C06981=1020.856,-123.857,-92.443,165.651,50.484,159.026
C06982=1020.861,-123.606,-92.451,165.655,50.481,159.026
C06983=1020.867,-123.357,-92.459,165.658,50.476,159.025
C06984=1020.872,-123.107,-92.467,165.660,50.472,159.025
C06985=1020.877,-122.857,-92.475,165.663,50.468,159.025
C06986=1020.883,-122.607,-92.482,165.667,50.464,159.025
C06987=1020.888,-122.357,-92.491,165.670,50.460,159.025
C06988=1020.893,-122.107,-92.499,165.673,50.456,159.025
C06989=1020.899,-121.857,-92.507,165.675,50.452,159.024
C06990=1020.904,-121.608,-92.515,165.679,50.448,159.024
C06991=1020.908,-121.358,-92.522,165.682,50.444,159.024
C06992=1020.914,-121.109,-92.530,165.685,50.440,159.024
C06993=1020.920,-120.859,-92.539,165.688,50.436,159.024
C06994=1020.925,-120.609,-92.547,165.691,50.431,159.023
C06995=1020.930,-120.359,-92.555,165.694,50.428,159.023
C06996=1020.936,-120.109,-92.562,165.697,50.424,159.023
C06997=1020.941,-119.859,-92.571,165.700,50.420,159.023
C06998=1020.946,-119.609,-92.579,165.703,50.415,159.023
C06999=1020.952,-119.359,-92.586,165.707,50.412,159.023
C07000=1020.957,-119.110,-92.595,165.709,50.408,159.022
C07001=1020.962,-118.860,-92.603,165.712,50.404,159.022
C07002=1020.967,-118.610,-92.611,165.716,50.399,159.022
C07003=1020.973,-118.360,-92.619,165.718,50.395,159.022
C07004=1020.979,-118.111,-92.627,165.721,50.392,159.022
C07005=1020.985,-117.826,-92.637,165.725,50.387,159.021
C07006=1020.991,-117.542,-92.646,165.729,50.382,159.021
C07007=1020.997,-117.257,-92.656,165.732,50.378,159.021
C07008=1021.003,-116.972,-92.665,165.736,50.373,159.021
C07009=1021.009,-116.722,-92.672,165.739,50.369,159.021
C07010=1021.014,-116.472,-92.681,165.741,50.365,159.021
C07011=1021.019,-116.222,-92.689,165.744,50.361,159.020
C07012=1021.025,-115.973,-92.698,165.748,50.357,159.020
C07013=1021.031,-115.723,-92.706,165.751,50.352,159.020
C07014=1021.036,-115.473,-92.714,165.754,50.349,159.020
C07015=1021.041,-115.223,-92.722,165.757,50.345,159.020
C07016=1021.046,-114.973,-92.731,165.760,50.341,159.019
C07017=1021.051,-114.724,-92.739,165.763,50.336,159.019
C07018=1021.057,-114.474,-92.747,165.765,50.332,159.019
C07019=1021.063,-114.225,-92.755,165.770,50.329,159.019
C07020=1021.068,-113.975,-92.764,165.772,50.325,159.019
C07021=1021.073,-113.724,-92.772,165.775,50.320,159.018
C07022=1021.079,-113.474,-92.781,165.778,50.317,159.018
C07023=1021.084,-113.224,-92.789,165.782,50.313,159.018
C07024=1021.089,-112.975,-92.797,165.785,50.308,159.018
C07025=1021.094,-112.725,-92.806,165.787,50.304,159.018
C07026=1021.100,-112.475,-92.814,165.790,50.301,159.018
C07027=1021.105,-112.226,-92.823,165.794,50.297,159.018
C07028=1021.111,-111.976,-92.831,165.797,50.292,159.017
C07029=1021.117,-111.726,-92.840,165.799,50.288,159.017
C07030=1021.122,-111.476,-92.848,165.803,50.285,159.017
C07031=1021.127,-111.226,-92.857,165.806,50.281,159.017
C07032=1021.133,-110.977,-92.865,165.809,50.276,159.017
C07033=1021.138,-110.727,-92.874,165.812,50.272,159.016
C07034=1021.143,-110.477,-92.882,165.815,50.269,159.016
C07035=1021.148,-110.227,-92.891,165.819,50.265,159.016
C07036=1021.154,-109.977,-92.899,165.821,50.260,159.016
C07037=1021.160,-109.727,-92.908,165.824,50.256,159.016
C07038=1021.165,-109.478,-92.916,165.827,50.252,159.015
C07039=1021.170,-109.228,-92.925,165.831,50.248,159.015
C07040=1021.176,-108.979,-92.933,165.833,50.244,159.015
C07041=1021.182,-108.729,-92.942,165.836,50.240,159.015
C07042=1021.188,-108.479,-92.951,165.840,50.236,159.015
C07043=1021.193,-108.229,-92.959,165.843,50.232,159.014
C07044=1021.198,-107.980,-92.968,165.846,50.228,159.014
C07045=1021.204,-107.729,-92.977,165.848,50.224,159.014
C07046=1021.209,-107.479,-92.985,165.852,50.220,159.014
C07047=1021.214,-107.230,-92.994,165.855,50.216,159.014
C07048=1021.220,-106.981,-93.003,165.858,50.212,159.014
C07049=1021.226,-106.730,-93.012,165.861,50.208,159.013
C07050=1021.231,-106.480,-93.020,165.864,50.204,159.013
C07051=1021.236,-106.231,-93.029,165.867,50.200,159.013
C07052=1021.241,-105.981,-93.038,165.870,50.196,159.013
C07053=1021.247,-105.731,-93.047,165.873,50.192,159.013
C07054=1021.252,-105.481,-93.056,165.877,50.188,159.012
C07055=1021.258,-105.231,-93.064,165.880,50.185,159.012
C07056=1021.263,-104.982,-93.073,165.882,50.180,159.012
C07057=1021.269,-104.732,-93.082,165.885,50.176,159.012
C07058=1021.274,-104.482,-93.091,165.889,50.172,159.012
C07059=1021.280,-104.233,-93.099,165.892,50.169,159.012
C07060=1021.286,-103.983,-93.109,165.895,50.164,159.011
C07061=1021.291,-103.733,-93.117,165.897,50.160,159.011
C07062=1021.296,-103.483,-93.126,165.901,50.156,159.011
C07063=1021.301,-103.233,-93.135,165.904,50.153,159.011
C07064=1021.307,-102.983,-93.144,165.907,50.148,159.011
C07065=1021.312,-102.734,-93.153,165.910,50.144,159.010
C07066=1021.318,-102.484,-93.163,165.913,50.140,159.010
C07067=1021.324,-102.234,-93.171,165.916,50.137,159.010
C07068=1021.329,-101.985,-93.179,165.919,50.133,159.010
C07069=1021.335,-101.700,-93.190,165.923,50.128,159.010
C07070=1021.342,-101.414,-93.200,165.926,50.123,159.009
C07071=1021.347,-101.130,-93.211,165.930,50.119,159.009
C07072=1021.354,-100.845,-93.221,165.933,50.115,159.009
C07073=1021.360,-100.546,-93.231,165.937,50.109,159.009
C07074=1021.367,-100.246,-93.242,165.941,50.105,159.009
C07075=1021.374,-99.946,-93.253,165.944,50.100,159.008
C07076=1021.381,-99.647,-93.264,165.948,50.095,159.008
C07077=1021.386,-99.397,-93.273,165.951,50.091,159.008
C07078=1021.391,-99.148,-93.283,165.954,50.087,159.008
C07079=1021.397,-98.898,-93.291,165.957,50.083,159.008
C07080=1021.403,-98.648,-93.301,165.960,50.079,159.007
C07081=1021.408,-98.398,-93.310,165.963,50.075,159.007
C07082=1021.414,-98.149,-93.319,165.967,50.071,159.007
C07083=1021.420,-97.898,-93.328,165.970,50.067,159.007
C07084=1021.425,-97.649,-93.337,165.972,50.063,159.007
C07085=1021.431,-97.399,-93.346,165.975,50.059,159.006
C07086=1021.435,-97.149,-93.356,165.978,50.055,159.006
C07087=1021.441,-96.900,-93.365,165.982,50.052,159.006
C07088=1021.447,-96.650,-93.374,165.985,50.047,159.006
C07089=1021.452,-96.400,-93.384,165.988,50.043,159.006
C07090=1021.458,-96.151,-93.393,165.991,50.040,159.006
C07091=1021.462,-95.901,-93.402,165.993,50.036,159.005
C07092=1021.469,-95.651,-93.412,165.998,50.032,159.005
C07093=1021.473,-95.401,-93.422,166.000,50.028,159.005
C07094=1021.480,-95.152,-93.431,166.003,50.024,159.005
C07095=1021.485,-94.902,-93.440,166.006,50.021,159.005
C07096=1021.490,-94.652,-93.450,166.009,50.017,159.004
C07097=1021.496,-94.403,-93.459,166.011,50.013,159.004
C07098=1021.501,-94.152,-93.469,166.016,50.009,159.004
C07099=1021.507,-93.903,-93.478,166.018,50.005,159.004
C07100=1021.512,-93.653,-93.488,166.021,50.001,159.004
C07101=1021.518,-93.404,-93.497,166.024,49.997,159.004
C07102=1021.523,-93.153,-93.506,166.028,49.993,159.003
C07103=1021.528,-92.904,-93.516,166.031,49.989,159.003
C07104=1021.534,-92.654,-93.525,166.034,49.986,159.003
C07105=1021.540,-92.404,-93.536,166.036,49.981,159.003
C07106=1021.545,-92.155,-93.545,166.039,49.977,159.003
C07107=1021.551,-91.904,-93.554,166.043,49.974,159.003
C07108=1021.556,-91.655,-93.563,166.046,49.970,159.002
C07109=1021.562,-91.405,-93.574,166.049,49.966,159.002
C07110=1021.567,-91.156,-93.583,166.051,49.962,159.002
C07111=1021.573,-90.906,-93.592,166.055,49.958,159.002
C07112=1021.579,-90.656,-93.603,166.058,49.954,159.002
C07113=1021.584,-90.406,-93.611,166.061,49.950,159.001
C07114=1021.589,-90.156,-93.621,166.064,49.946,159.001
C07115=1021.595,-89.907,-93.630,166.067,49.942,159.001
C07116=1021.600,-89.657,-93.641,166.071,49.938,159.001
C07117=1021.607,-89.407,-93.650,166.073,49.934,159.001
C07118=1021.611,-89.158,-93.660,166.076,49.930,159.000
C07119=1021.618,-88.908,-93.670,166.079,49.926,159.000
C07120=1021.623,-88.658,-93.680,166.082,49.922,159.000
C07121=1021.629,-88.409,-93.689,166.086,49.919,159.000
C07122=1021.634,-88.158,-93.698,166.089,49.915,159.000
C07123=1021.640,-87.908,-93.708,166.091,49.911,158.999
C07124=1021.645,-87.659,-93.717,166.094,49.906,158.999
C07125=1021.651,-87.409,-93.727,166.098,49.903,158.999
C07126=1021.657,-87.159,-93.737,166.101,49.899,158.999
C07127=1021.662,-86.910,-93.747,166.104,49.895,158.999
C07128=1021.668,-86.660,-93.756,166.106,49.891,158.998
C07129=1021.673,-86.419,-93.766,166.109,49.887,158.998
C07130=1021.679,-86.177,-93.775,166.113,49.883,158.998
C07131=1021.684,-85.936,-93.785,166.116,49.879,158.998
C07132=1021.690,-85.695,-93.794,166.119,49.876,158.998
C07133=1021.696,-85.453,-93.804,166.122,49.871,158.997
C07134=1021.701,-85.212,-93.813,166.125,49.867,158.997
C07135=1021.706,-84.970,-93.823,166.128,49.864,158.997
C07136=1021.711,-84.729,-93.832,166.130,49.860,158.997
C07137=1021.717,-84.479,-93.842,166.133,49.856,158.997
C07138=1021.723,-84.229,-93.851,166.137,49.852,158.996
C07139=1021.728,-83.980,-93.861,166.140,49.848,158.996
C07140=1021.735,-83.730,-93.871,166.143,49.844,158.996
C07141=1021.740,-83.480,-93.881,166.145,49.840,158.996
C07142=1021.746,-83.230,-93.890,166.149,49.836,158.996
C07143=1021.751,-82.981,-93.901,166.152,49.832,158.995
C07144=1021.757,-82.732,-93.910,166.155,49.828,158.995
C07145=1021.763,-82.482,-93.921,166.158,49.824,158.995
C07146=1021.769,-82.232,-93.930,166.161,49.820,158.995
C07147=1021.774,-81.982,-93.940,166.164,49.816,158.994
C07148=1021.780,-81.733,-93.950,166.167,49.812,158.994
C07149=1021.785,-81.482,-93.960,166.170,49.808,158.994
C07150=1021.792,-81.233,-93.969,166.173,49.803,158.994
C07151=1021.797,-80.983,-93.980,166.177,49.800,158.994
C07152=1021.804,-80.733,-93.990,166.179,49.796,158.993
C07153=1021.809,-80.483,-94.000,166.183,49.792,158.993
C07154=1021.815,-80.234,-94.009,166.186,49.788,158.993
C07155=1021.820,-79.984,-94.019,166.188,49.784,158.993
C07156=1021.826,-79.735,-94.030,166.192,49.780,158.993
C07157=1021.831,-79.484,-94.040,166.194,49.776,158.992
C07158=1021.837,-79.235,-94.050,166.198,49.772,158.992
C07159=1021.843,-78.985,-94.061,166.201,49.768,158.992
C07160=1021.848,-78.735,-94.071,166.204,49.764,158.992
C07161=1021.853,-78.486,-94.081,166.207,49.760,158.992
C07162=1021.860,-78.236,-94.091,166.210,49.757,158.991
C07163=1021.865,-77.986,-94.101,166.212,49.753,158.991
C07164=1021.871,-77.736,-94.111,166.216,49.749,158.991
C07165=1021.876,-77.487,-94.122,166.219,49.745,158.991
C07166=1021.882,-77.237,-94.132,166.222,49.741,158.991
C07167=1021.888,-76.987,-94.142,166.225,49.737,158.990
C07168=1021.894,-76.737,-94.153,166.227,49.733,158.990
C07169=1021.899,-76.488,-94.163,166.232,49.729,158.990
C07170=1021.904,-76.238,-94.173,166.234,49.725,158.990
C07171=1021.911,-75.989,-94.183,166.237,49.721,158.989
C07172=1021.916,-75.739,-94.194,166.240,49.717,158.989
C07173=1021.922,-75.489,-94.204,166.243,49.714,158.989
C07174=1021.927,-75.239,-94.214,166.247,49.710,158.989
C07175=1021.933,-74.989,-94.225,166.249,49.706,158.989
C07176=1021.939,-74.740,-94.235,166.252,49.702,158.988
C07177=1021.945,-74.490,-94.246,166.255,49.698,158.988
C07178=1021.950,-74.240,-94.256,166.258,49.694,158.988
C07179=1021.956,-73.991,-94.267,166.261,49.690,158.988
C07180=1021.961,-73.740,-94.277,166.265,49.687,158.988
C07181=1021.967,-73.491,-94.288,166.268,49.682,158.987
C07182=1021.973,-73.241,-94.299,166.271,49.679,158.987
C07183=1021.978,-72.991,-94.309,166.273,49.675,158.987
C07184=1021.984,-72.742,-94.320,166.277,49.672,158.987
C07185=1021.989,-72.492,-94.331,166.279,49.668,158.987
C07186=1021.994,-72.242,-94.341,166.282,49.664,158.987
C07187=1022.000,-71.992,-94.352,166.285,49.660,158.986
C07188=1022.006,-71.743,-94.363,166.288,49.656,158.986
